// TwinCAT 3 PLC project CNM_AssertionInterfaceTests
// Title: CNM_AssertionInterfaceTests
// Company: ekvip automation GmbH
// Author: boez & ajum
// ProjectVersion: 1.2.0.6
// Description: dirty desperate Foo bar baz run it or go to jail
// ProgramVersion: 3.1.4026.19
// libraries:
//   CNM_AbstractObject, * (ekvip automation GmbH)
//   CNM_AssertionInterfaces, * (ekvip automation GmbH)
//   CNM_ReturnTypes, * (ekvip automation GmbH)
//   CNM_UnicodeUtilities, * (ekvip automation GmbH)
//   Tc2_CncBase, * (Beckhoff Automation GmbH)
//   Tc2_CncHli, * (Beckhoff Automation GmbH)
//   Tc2_Standard, * (Beckhoff Automation GmbH)
//   Tc2_System, * (Beckhoff Automation GmbH)
//   Tc2_Utilities, * (Beckhoff Automation GmbH)
//   Tc3_Module, * (Beckhoff Automation GmbH)
//   TcUnit, * (www.tcunit.org)
// project tree:
//   AssertionTester/AssertionResult/interfaces/ IAssertorContainer.TcIO
//   AssertionTester/AssertionTests/BinaryAssertions/classes/ BinaryAssertionsTests.TcPOU
//   AssertionTester/AssertionTests/BitNumberAssertions/classes/ ByteAssertionTests.TcPOU, XWordAssertionTests.TcPOU, LWordAssertionTests.TcPOU, DWordAssertionTests.TcPOU, WordAssertionTests.TcPOU, XWordAssertionTests.TcPOU
//   AssertionTester/AssertionTests/classes/ AbstractAssertorTest.TcPOU
//   AssertionTester/AssertionTests/DateTimeAssertions/classes/ DTAssertionTests.TcPOU, DateAssertionTests.TcPOU, LDateAssertionTests.TcPOU, LDTAssertionTests.TcPOU, LTODAssertionTests.TcPOU, TODAssertionTests.TcPOU
//   AssertionTester/AssertionTests/FloatAssertions/classes/ LRealAssertionTests.TcPOU, RealAssertionTests.TcPOU
//   AssertionTester/AssertionTests/FloatAssertions/types/structs/ LRealTestParameter.TcDUT (not stored)
//   AssertionTester/AssertionTests/IntegerAssertions/classes/ DintAssertionTests.TcPOU, IntAssertionTests.TcPOU, LintAssertionTests.TcPOU, SintAssertionTests.TcPOU, UdintAssertionTests.TcPOU, UintAssertionTests.TcPOU, UlintAssertionTests.TcPOU, UsintAssertionTests.TcPOU, UxintAssertionTests.TcPOU, XintAssertionTests.TcPOU
//   AssertionTester/AssertionTests/ObjectAssertions/classes/internal/ ConcreteObject.TcPOU, DWordValue.TcPOU, ReverseOrderComparator.TcPOU
//   AssertionTester/AssertionTests/ObjectAssertions/classes/ ObjectAssertionsTests.TcPOU
//   AssertionTester/AssertionTests/ObjectAssertions/interfaces/ IDWord.TcIO
//   AssertionTester/AssertionTests/PointerAssertions/classes/ PointerAssertionsTests.TcPOU
//   AssertionTester/AssertionTests/StringAssertions/classes/ UnicodeUtf16StringAssertionTests.TcPOU, UnicodeUtf8StringAssertionTests.TcPOU, Windows125xStringAssertionTests.TcPOU
//   AssertionTester/AssertionTests/TimeAssertions/classes/ LTimeAssertionsTests.TcPOU, TimeAssertionsTests.TcPOU
//   AssertionTester/classes/ AssertionTester.TcPOU
//   AssertionTester/interfaces/ IAttachAssertorContainer.TcIO
//   Project Information/ F_GetCompany.TcPOU, F_GetTitle.TcPOU, F_GetVersion.TcPOU
//   Version/ Global_Version.TcGVL

// ---- Version/Global_Version.TcGVL
{attribute 'TcGenerated'}
{attribute 'no-analysis'}
{attribute 'linkalways'}
// This function has been automatically generated from the project information.
VAR_GLOBAL CONSTANT
	{attribute 'const_non_replaced'}
	stLibVersion_CNM_AssertionInterfaceTests : ST_LibVersion := (iMajor := 1, iMinor := 2, iBuild := 0, iRevision := 6, nFlags := 0, sVersion := '1.2.0.6');
END_VAR

// ---- AssertionTester/AssertionResult/interfaces/IAssertorContainer.TcIO
(*

short summary
=============
An assertion is handled internally, and there is no common way to determine if an assertion was wrong.
This interface is just a helper to build containers to test assertions in a unified way.

.. <legal notes>

legal notes
=================
| SPDX-FileCopyrightText: © 2023 ekvip automation GmbH <info@ekvip.de>
| SPDX-License-Identifier: Apache-2.0
| For details check: Apache-2.0_

.. _Apache-2.0: https://www.apache.org/licenses/LICENSE-2.0

.. </legal notes>

properties
==========

*)

INTERFACE IAssertorContainer //EXTENDS CNM_AbstractObject.IObject

PROPERTY assertor :CNM_AssertionInterfaces.IAssertor
GET
END_GET
END_PROPERTY

METHOD resetAssertor
VAR_INPUT
END_VAR
END_METHOD

(*

short summary
=============
This property is used by the tests to determine if the assertion was right or wrong (getter)

.. <legal notes>

legal notes
=================
| SPDX-FileCopyrightText: © 2022 ekvip automation GmbH <info@ekvip.de>
| SPDX-License-Identifier: Apache-2.0
| For details check: Apache-2.0_

.. _Apache-2.0: https://www.apache.org/licenses/LICENSE-2.0

.. </legal notes>

*)

PROPERTY wasAssertionWrong :BOOL
GET
END_GET
END_PROPERTY

END_INTERFACE

// ---- AssertionTester/AssertionTests/ObjectAssertions/interfaces/IDWord.TcIO
(*

short summary
=============
Interface for DWordValue Class
only needed for ´´__QUERYINTERFACE()´´ in ´´compareTo()´´
.. <legal notes>

legal notes
=================
| SPDX-FileCopyrightText: © 2023 ekvip automation GmbH <info@ekvip.de>
| SPDX-License-Identifier: Apache-2.0
| For details check: Apache-2.0_

.. _Apache-2.0: https://www.apache.org/licenses/LICENSE-2.0

.. </legal notes>

*)

INTERFACE IDWord EXTENDS CNM_AbstractObject.IObject

(*

short summary
=============
value of the DWordValue Class

.. <legal notes>

legal notes
=================
| SPDX-FileCopyrightText: © 2023 ekvip automation GmbH <info@ekvip.de>
| SPDX-License-Identifier: Apache-2.0
| For details check: Apache-2.0_

.. _Apache-2.0: https://www.apache.org/licenses/LICENSE-2.0

.. </legal notes>

*)

PROPERTY value : DWORD
GET
END_GET
SET
END_SET
END_PROPERTY

END_INTERFACE

// ---- AssertionTester/interfaces/IAttachAssertorContainer.TcIO
(*

short summary
=============

.. <legal notes>

legal notes
=================
| SPDX-FileCopyrightText: © 2023 ekvip automation GmbH <info@ekvip.de>
| SPDX-License-Identifier: Apache-2.0
| For details check: Apache-2.0_

.. _Apache-2.0: https://www.apache.org/licenses/LICENSE-2.0

.. </legal notes>

*)

INTERFACE IAttachAssertorContainer EXTENDS  __SYSTEM.IQueryInterface

(*

short summary
=============

.. <legal notes>

legal notes
=================
| SPDX-FileCopyrightText: © 2023 ekvip automation GmbH <info@ekvip.de>
| SPDX-License-Identifier: Apache-2.0
| For details check: Apache-2.0_

.. _Apache-2.0: https://www.apache.org/licenses/LICENSE-2.0

.. </legal notes>

*)

PROPERTY attachAssertorContainer : IAssertorContainer
SET
END_SET
END_PROPERTY

END_INTERFACE

// ---- AssertionTester/AssertionTests/BinaryAssertions/classes/BinaryAssertionsTests.TcPOU
(*

short summary
==================
This class tests all methods of binary assertions
with various combinations of inputs and checks expected 
outputs are satisfied or not

.. <legal notes>

legal notes
=================
| SPDX-FileCopyrightText: © 2022 ekvip automation GmbH <info@ekvip.de>
| SPDX-License-Identifier: Apache-2.0
| For details check: Apache-2.0_

.. _Apache-2.0: https://www.apache.org/licenses/LICENSE-2.0

.. </legal notes>

methods and properties
======================

*)

FUNCTION_BLOCK BinaryAssertionsTests EXTENDS AbstractAssertorTest
VAR_INPUT
	(* shall be not set, because this is for the null pointer edge case tests *)
	NULL :ANY;
END_VAR
VAR
	(* boolean value TRUE *)
	BOOLEAN_TRUE							:BOOL := TRUE;
	(* boolean value FALSE *)
	BOOLEAN_FALSE							:BOOL := FALSE;
	(* long word value one *)
	LWORD_WITH_VALUE_1						:LWORD := 16#0000_0000_0000_0000_0000_0000_0000_0001;
	(* word value 255 *)
	ALL_BITS_SET_AT_LOW_BYTE				:WORD := 16#00FF;
	(* double word vaule 255 *)
	ALL_BITS_SET_AT_LOW_BYTE_DWORD			:DWORD := 16#0000_00FF;
	(* double word value 16#FF00_FF00 *)
	NO_BITS_SET_AT_MID_BYTES				:DWORD := 16#FF00_00FF;
	(* byte array [0..299] all zero *)
	BYTE_ARRAY_ALL_BYTES_ZERO				:ARRAY[0..299] OF BYTE := [300(0)];
	(* byte array [0..299] 100 zero, 100 16#FF, 100 zero *)
	BYTE_ARRAY_MID_BYTES_FF_ONLY			:ARRAY[0..299] OF BYTE := [100(0),100(16#FF),100(0)];
	(* byte array with two dimensions [0..2][0..99] all zero *)
	ARRAY_OF_BYTE_ARRAY_ALL_BYTES_ZERO		:ARRAY[0..2] OF ARRAY[0..99] OF BYTE := [[100(0)],[100(0)],[100(0)]];	
END_VAR
VAR CONSTANT	
	(* prefix to unify the test names *)
	TEST_NAME_PREFIX						:STRING := 'assert.binary.';
END_VAR

THIS^.runIsEqualToTests();
THIS^.runIsNotEqualToTests();
THIS^.runIsGreaterThanTests();
THIS^.runIsLessThanTests();

(*

short summary
==================
This test method is a helper function to create a unified test name

.. <legal notes>

legal notes
=================
| SPDX-FileCopyrightText: © 2022 ekvip automation GmbH <info@ekvip.de>
| SPDX-License-Identifier: Apache-2.0
| For details check: Apache-2.0_

.. _Apache-2.0: https://www.apache.org/licenses/LICENSE-2.0

.. </legal notes>

parameters
==========

*)

METHOD PROTECTED getTestNameFor :Tc2_System.T_MaxString
VAR_INPUT
	(* name of the method to test, to create a unified test name *)
	nameOfMethodToTest	:Tc2_System.T_MaxString;
END_VAR
getTestNameFor := Tc2_Standard.CONCAT(THIS^.TEST_NAME_PREFIX, nameOfMethodToTest);
END_METHOD

(*

short summary
==================
This test method tests ``assert.binary.isEqualTo``
method of CNM_AssertionInterfaces library with various inputs

.. <legal notes>

legal notes
=================
| SPDX-FileCopyrightText: © 2022 ekvip automation GmbH <info@ekvip.de>
| SPDX-License-Identifier: Apache-2.0
| For details check: Apache-2.0_

.. _Apache-2.0: https://www.apache.org/licenses/LICENSE-2.0

.. </legal notes>

*)

METHOD runIsEqualToTests
RETURN (NOT TcUnit.TEST_ORDERED(THIS^.getTestNameFor('isEqualTo')));

THIS^.testIsEqualTo(
	data			:= THIS^.BOOLEAN_FALSE,
	dataToCompare	:= THIS^.BOOLEAN_FALSE,
	assertionIsWrong:= FALSE,
	testDataInfo	:= 'data is a boolean FALSE, dataToCompare is a aboolean FALSE'
);

THIS^.testIsEqualTo(
	data			:= THIS^.BOOLEAN_TRUE,
	dataToCompare	:= THIS^.BOOLEAN_FALSE,
	assertionIsWrong:= TRUE,
	testDataInfo	:= 'data is a boolean TRUE, dataToCompare is a boolean FALSE'
);

THIS^.testIsEqualTo(
	data			:= THIS^.BOOLEAN_TRUE,
	dataToCompare	:= NULL,
	assertionIsWrong:= TRUE,
	testDataInfo	:= 'data is a boolean TRUE, dataToCompare is null'
);

THIS^.testIsEqualTo(
	data			:= NULL,
	dataToCompare	:= NULL,
	assertionIsWrong:= FALSE,
	testDataInfo	:= 'data is null, dataToCompare is null'
);

THIS^.testIsEqualTo(
	data			:= THIS^.BYTE_ARRAY_ALL_BYTES_ZERO,
	dataToCompare	:= THIS^.BOOLEAN_FALSE,
	assertionIsWrong:= FALSE,
	testDataInfo	:= 'data is a byte array [300(0)], dataToCompare is a boolean FALSE'
);

THIS^.testIsEqualTo(
	data			:= THIS^.BYTE_ARRAY_ALL_BYTES_ZERO,
	dataToCompare	:= THIS^.ARRAY_OF_BYTE_ARRAY_ALL_BYTES_ZERO,
	assertionIsWrong:= FALSE,
	testDataInfo	:= 'data is a byte array [300(0)], dataToCompare is a byte array [[100(0)],[100(0)],[100(0)]]'
);

THIS^.testIsEqualTo(
	data			:= THIS^.BYTE_ARRAY_MID_BYTES_FF_ONLY,
	dataToCompare	:= THIS^.ARRAY_OF_BYTE_ARRAY_ALL_BYTES_ZERO,
	assertionIsWrong:= TRUE,
	testDataInfo	:= 'data is a byte array [100(0),100(16#FF),100(0)], dataToCompare is a byte array [[100(0)],[100(0)],[100(0)]]'
);

THIS^.testIsEqualTo(
	data			:= THIS^.ALL_BITS_SET_AT_LOW_BYTE,
	dataToCompare	:= THIS^.ALL_BITS_SET_AT_LOW_BYTE_DWORD,
	assertionIsWrong:= FALSE,
	testDataInfo	:= 'data is a word 16#00FF, dataToCompare is dword 16#0000_00FF'
);

THIS^.testIsEqualTo(
	data			:= THIS^.ALL_BITS_SET_AT_LOW_BYTE_DWORD,
	dataToCompare	:= THIS^.ALL_BITS_SET_AT_LOW_BYTE,
	assertionIsWrong:= FALSE,
	testDataInfo	:= 'data is a dword 16#0000_00FF, dataToCompare is word 16#00FF'
);

THIS^.testIsEqualTo(
	data			:= THIS^.ALL_BITS_SET_AT_LOW_BYTE,
	dataToCompare	:= THIS^.NO_BITS_SET_AT_MID_BYTES,
	assertionIsWrong:= TRUE,
	testDataInfo	:= 'data is a word 16#00FF, dataToCompare is dword 16#FF00_00FF'
);

THIS^.testIsEqualTo(
	data			:= THIS^.NO_BITS_SET_AT_MID_BYTES,
	dataToCompare	:= THIS^.ALL_BITS_SET_AT_LOW_BYTE,
	assertionIsWrong:= TRUE,
	testDataInfo	:= 'data is a dword 16#FF00_00FF, dataToCompare is word 16#00FF'
);

THIS^.testIsEqualTo(
	data			:= THIS^.LWORD_WITH_VALUE_1,
	dataToCompare	:= THIS^.BOOLEAN_TRUE,
	assertionIsWrong:= FALSE,
	testDataInfo	:= 'data is a lword 16#0000_0000_0000_0000_0000_0000_0000_0001, dataToCompare is bool TRUE'
);

THIS^.testIsEqualTo(
	data			:= THIS^.LWORD_WITH_VALUE_1,
	dataToCompare	:= THIS^.BOOLEAN_FALSE,
	assertionIsWrong:= TRUE,
	testDataInfo	:= 'data is a lword 16#0000_0000_0000_0000_0000_0000_0000_0001, dataToCompare is bool FALSE'
);

TcUnit.TEST_FINISHED();
END_METHOD

(*

short summary
==================
This test method tests ``assert.binary.isGreaterThan``
method of CNM_AssertionInterfaces library with various inputs

.. <legal notes>

legal notes
=================
| SPDX-FileCopyrightText: © 2022 ekvip automation GmbH <info@ekvip.de>
| SPDX-License-Identifier: Apache-2.0
| For details check: Apache-2.0_

.. _Apache-2.0: https://www.apache.org/licenses/LICENSE-2.0

.. </legal notes>

*)

METHOD runIsGreaterThanTests
RETURN (NOT TcUnit.TEST_ORDERED(THIS^.getTestNameFor('isGreaterThan')));

THIS^.testIsGreaterThan(
	data			:= THIS^.BOOLEAN_FALSE,
	dataToCompare	:= THIS^.BOOLEAN_FALSE,
	assertionIsWrong:= TRUE,
	testDataInfo	:= 'data is a boolean FALSE, dataToCompare is a aboolean FALSE'
);

THIS^.testIsGreaterThan(
	data			:= THIS^.BOOLEAN_TRUE,
	dataToCompare	:= THIS^.BOOLEAN_FALSE,
	assertionIsWrong:= FALSE,
	testDataInfo	:= 'data is a boolean TRUE, dataToCompare is a boolean FALSE'
);

THIS^.testIsGreaterThan(
	data			:= THIS^.BOOLEAN_TRUE,
	dataToCompare	:= NULL,
	assertionIsWrong:= FALSE,
	testDataInfo	:= 'data is a boolean TRUE, dataToCompare is null'
);

THIS^.testIsGreaterThan(
	data			:= NULL,
	dataToCompare	:= NULL,
	assertionIsWrong:= TRUE,
	testDataInfo	:= 'data is null, dataToCompare is null'
);

THIS^.testIsGreaterThan(
	data			:= THIS^.BYTE_ARRAY_ALL_BYTES_ZERO,
	dataToCompare	:= THIS^.BOOLEAN_FALSE,
	assertionIsWrong:= TRUE,
	testDataInfo	:= 'data is a byte array [300(0)], dataToCompare is a boolean FALSE'
);

THIS^.testIsGreaterThan(
	data			:= THIS^.BYTE_ARRAY_ALL_BYTES_ZERO,
	dataToCompare	:= THIS^.ARRAY_OF_BYTE_ARRAY_ALL_BYTES_ZERO,
	assertionIsWrong:= TRUE,
	testDataInfo	:= 'data is a byte array [300(0)], dataToCompare is a byte array [[100(0)],[100(0)],[100(0)]]'
);

THIS^.testIsGreaterThan(
	data			:= THIS^.BYTE_ARRAY_MID_BYTES_FF_ONLY,
	dataToCompare	:= THIS^.ARRAY_OF_BYTE_ARRAY_ALL_BYTES_ZERO,
	assertionIsWrong:= FALSE,
	testDataInfo	:= 'data is a byte array [100(0),100(16#FF),100(0)], dataToCompare is a byte array [[100(0)],[100(0)],[100(0)]]'
);

THIS^.testIsGreaterThan(
	data			:= THIS^.ALL_BITS_SET_AT_LOW_BYTE,
	dataToCompare	:= THIS^.ALL_BITS_SET_AT_LOW_BYTE_DWORD,
	assertionIsWrong:= TRUE,
	testDataInfo	:= 'data is a word 16#00FF, dataToCompare is dword 16#0000_00FF'
);

THIS^.testIsGreaterThan(
	data			:= THIS^.ALL_BITS_SET_AT_LOW_BYTE_DWORD,
	dataToCompare	:= THIS^.ALL_BITS_SET_AT_LOW_BYTE,
	assertionIsWrong:= TRUE,
	testDataInfo	:= 'data is a dword 16#0000_00FF, dataToCompare is word 16#00FF'
);

THIS^.testIsGreaterThan(
	data			:= THIS^.ALL_BITS_SET_AT_LOW_BYTE,
	dataToCompare	:= THIS^.NO_BITS_SET_AT_MID_BYTES,
	assertionIsWrong:= TRUE,
	testDataInfo	:= 'data is a word 16#00FF, dataToCompare is dword 16#FF00_00FF'
);

THIS^.testIsGreaterThan(
	data			:= THIS^.NO_BITS_SET_AT_MID_BYTES,
	dataToCompare	:= THIS^.ALL_BITS_SET_AT_LOW_BYTE,
	assertionIsWrong:= FALSE,
	testDataInfo	:= 'data is a dword 16#FF00_00FF, dataToCompare is word 16#00FF'
);

THIS^.testIsGreaterThan(
	data			:= THIS^.LWORD_WITH_VALUE_1,
	dataToCompare	:= THIS^.BOOLEAN_TRUE,
	assertionIsWrong:= TRUE,
	testDataInfo	:= 'data is a lword 16#0000_0000_0000_0000_0000_0000_0000_0001, dataToCompare is bool TRUE'
);

THIS^.testIsGreaterThan(
	data			:= THIS^.LWORD_WITH_VALUE_1,
	dataToCompare	:= THIS^.BOOLEAN_FALSE,
	assertionIsWrong:= FALSE,
	testDataInfo	:= 'data is a lword 16#0000_0000_0000_0000_0000_0000_0000_0001, dataToCompare is bool FALSE'
);

THIS^.testIsGreaterThan(
	data			:= THIS^.BOOLEAN_TRUE,
	dataToCompare	:= THIS^.LWORD_WITH_VALUE_1,
	assertionIsWrong:= TRUE,
	testDataInfo	:= 'data is a bool TRUE, dataToCompare is bool 16#0000_0000_0000_0000_0000_0000_0000_0001'
);

THIS^.testIsGreaterThan(
	data			:= THIS^.BOOLEAN_FALSE,
	dataToCompare	:= THIS^.LWORD_WITH_VALUE_1,
	assertionIsWrong:= TRUE,
	testDataInfo	:= 'data is a bool FALSE, dataToCompare is bool 16#0000_0000_0000_0000_0000_0000_0000_0001'
);

TcUnit.TEST_FINISHED();
END_METHOD

(*

short summary
==================
This test method tests ``assert.binary.isLessThan``
method of CNM_AssertionInterfaces library with various inputs

.. <legal notes>

legal notes
=================
| SPDX-FileCopyrightText: © 2022 ekvip automation GmbH <info@ekvip.de>
| SPDX-License-Identifier: Apache-2.0
| For details check: Apache-2.0_

.. _Apache-2.0: https://www.apache.org/licenses/LICENSE-2.0

.. </legal notes>

*)

METHOD runIsLessThanTests
RETURN (NOT TcUnit.TEST_ORDERED(THIS^.getTestNameFor('isLessThan')));

THIS^.testIsLessThan(
	data			:= THIS^.BOOLEAN_FALSE,
	dataToCompare	:= THIS^.BOOLEAN_FALSE,
	assertionIsWrong:= TRUE,
	testDataInfo	:= 'data is a boolean FALSE, dataToCompare is a aboolean FALSE'
);

THIS^.testIsLessThan(
	data			:= THIS^.BOOLEAN_TRUE,
	dataToCompare	:= THIS^.BOOLEAN_FALSE,
	assertionIsWrong:= TRUE,
	testDataInfo	:= 'data is a boolean TRUE, dataToCompare is a boolean FALSE'
);

THIS^.testIsLessThan(
	data			:= THIS^.BOOLEAN_FALSE,
	dataToCompare	:= THIS^.BOOLEAN_TRUE,
	assertionIsWrong:= FALSE,
	testDataInfo	:= 'data is a boolean FALSE, dataToCompare is a boolean TRUE'
);

THIS^.testIsLessThan(
	data			:= THIS^.BOOLEAN_TRUE,
	dataToCompare	:= NULL,
	assertionIsWrong:= TRUE,
	testDataInfo	:= 'data is a boolean TRUE, dataToCompare is null'
);

THIS^.testIsLessThan(
	data			:= NULL,
	dataToCompare	:= THIS^.BOOLEAN_TRUE,
	assertionIsWrong:= FALSE,
	testDataInfo	:= 'data is null, dataToCompare is a boolean TRUE'
);

THIS^.testIsLessThan(
	data			:= NULL,
	dataToCompare	:= NULL,
	assertionIsWrong:= TRUE,
	testDataInfo	:= 'data is null, dataToCompare is null'
);

THIS^.testIsLessThan(
	data			:= THIS^.BYTE_ARRAY_ALL_BYTES_ZERO,
	dataToCompare	:= THIS^.BOOLEAN_FALSE,
	assertionIsWrong:= TRUE,
	testDataInfo	:= 'data is a byte array [300(0)], dataToCompare is a boolean FALSE'
);

THIS^.testIsLessThan(
	data			:= THIS^.BYTE_ARRAY_ALL_BYTES_ZERO,
	dataToCompare	:= THIS^.ARRAY_OF_BYTE_ARRAY_ALL_BYTES_ZERO,
	assertionIsWrong:= TRUE,
	testDataInfo	:= 'data is a byte array [300(0)], dataToCompare is a byte array [[100(0)],[100(0)],[100(0)]]'
);

THIS^.testIsLessThan(
	data			:= THIS^.ARRAY_OF_BYTE_ARRAY_ALL_BYTES_ZERO,
	dataToCompare	:= THIS^.BYTE_ARRAY_ALL_BYTES_ZERO,
	assertionIsWrong:= TRUE,
	testDataInfo	:= 'data is a byte array [100(0),100(0),100(0)], dataToCompare is a byte array [300(0)]'
);

THIS^.testIsLessThan(
	data			:= THIS^.BYTE_ARRAY_MID_BYTES_FF_ONLY,
	dataToCompare	:= THIS^.ARRAY_OF_BYTE_ARRAY_ALL_BYTES_ZERO,
	assertionIsWrong:= TRUE,
	testDataInfo	:= 'data is a byte array [100(0),100(16#FF),100(0)], dataToCompare is a byte array [[100(0)],[100(0)],[100(0)]]'
);

THIS^.testIsLessThan(
	data			:= THIS^.ARRAY_OF_BYTE_ARRAY_ALL_BYTES_ZERO,
	dataToCompare	:= THIS^.BYTE_ARRAY_MID_BYTES_FF_ONLY,
	assertionIsWrong:= FALSE,
	testDataInfo	:= 'data is a byte array [[100(0)],[100(0)],[100(0)]], dataToCompare is a byte array [100(0),100(16#FF),100(0)]'
);

THIS^.testIsLessThan(
	data			:= THIS^.ALL_BITS_SET_AT_LOW_BYTE_DWORD,
	dataToCompare	:= THIS^.ALL_BITS_SET_AT_LOW_BYTE,
	assertionIsWrong:= TRUE,
	testDataInfo	:= 'data is a dword 16#0000_00FF, dataToCompare is word 16#00FF'
);

THIS^.testIsLessThan(
	data			:= THIS^.ALL_BITS_SET_AT_LOW_BYTE,
	dataToCompare	:= THIS^.NO_BITS_SET_AT_MID_BYTES,
	assertionIsWrong:= FALSE,
	testDataInfo	:= 'data is a word 16#00FF, dataToCompare is dword 16#FF00_00FF'
);

THIS^.testIsLessThan(
	data			:= THIS^.NO_BITS_SET_AT_MID_BYTES,
	dataToCompare	:= THIS^.ALL_BITS_SET_AT_LOW_BYTE,
	assertionIsWrong:= TRUE,
	testDataInfo	:= 'data is a dword 16#FF00_00FF, dataToCompare is word 16#00FF'
);

THIS^.testIsLessThan(
	data			:= THIS^.LWORD_WITH_VALUE_1,
	dataToCompare	:= THIS^.BOOLEAN_TRUE,
	assertionIsWrong:= TRUE,
	testDataInfo	:= 'data is a lword 16#0000_0000_0000_0000_0000_0000_0000_0001, dataToCompare is bool TRUE'
);

THIS^.testIsLessThan(
	data			:= THIS^.LWORD_WITH_VALUE_1,
	dataToCompare	:= THIS^.BOOLEAN_FALSE,
	assertionIsWrong:= TRUE,
	testDataInfo	:= 'data is a lword 16#0000_0000_0000_0000_0000_0000_0000_0001, dataToCompare is bool FALSE'
);

THIS^.testIsLessThan(
	data			:= THIS^.BOOLEAN_TRUE,
	dataToCompare	:= THIS^.LWORD_WITH_VALUE_1,
	assertionIsWrong:= TRUE,
	testDataInfo	:= 'data is a bool TRUE, dataToCompare is bool 16#0000_0000_0000_0000_0000_0000_0000_0001'
);

THIS^.testIsLessThan(
	data			:= THIS^.BOOLEAN_FALSE,
	dataToCompare	:= THIS^.LWORD_WITH_VALUE_1,
	assertionIsWrong:= FALSE,
	testDataInfo	:= 'data is a bool FALSE, dataToCompare is bool 16#0000_0000_0000_0000_0000_0000_0000_0001'
);

TcUnit.TEST_FINISHED();
END_METHOD

(*

short summary
==================
This test method tests ``assert.binary.isNotEqualTo``
method of CNM_AssertionInterfaces library with various inputs

.. <legal notes>

legal notes
=================
| SPDX-FileCopyrightText: © 2022 ekvip automation GmbH <info@ekvip.de>
| SPDX-License-Identifier: Apache-2.0
| For details check: Apache-2.0_

.. _Apache-2.0: https://www.apache.org/licenses/LICENSE-2.0

.. </legal notes>

*)

METHOD runIsNotEqualToTests
RETURN (NOT TcUnit.TEST_ORDERED(THIS^.getTestNameFor('isNotEqualTo')));

THIS^.testIsNotEqualTo(
	data			:= THIS^.BOOLEAN_FALSE,
	dataToCompare	:= THIS^.BOOLEAN_FALSE,
	assertionIsWrong:= TRUE,
	testDataInfo	:= 'data is a boolean FALSE, dataToCompare is a aboolean FALSE'
);

THIS^.testIsNotEqualTo(
	data			:= THIS^.BOOLEAN_TRUE,
	dataToCompare	:= THIS^.BOOLEAN_FALSE,
	assertionIsWrong:= FALSE,
	testDataInfo	:= 'data is a boolean TRUE, dataToCompare is a boolean FALSE'
);

THIS^.testIsNotEqualTo(
	data			:= THIS^.BOOLEAN_TRUE,
	dataToCompare	:= NULL,
	assertionIsWrong:= FALSE,
	testDataInfo	:= 'data is a boolean TRUE, dataToCompare is null'
);

THIS^.testIsNotEqualTo(
	data			:= NULL,
	dataToCompare	:= NULL,
	assertionIsWrong:= TRUE,
	testDataInfo	:= 'data is null, dataToCompare is null'
);

THIS^.testIsNotEqualTo(
	data			:= THIS^.BYTE_ARRAY_ALL_BYTES_ZERO,
	dataToCompare	:= THIS^.BOOLEAN_FALSE,
	assertionIsWrong:= TRUE,
	testDataInfo	:= 'data is a byte array [300(0)], dataToCompare is a boolean FALSE'
);

THIS^.testIsNotEqualTo(
	data			:= THIS^.BYTE_ARRAY_ALL_BYTES_ZERO,
	dataToCompare	:= THIS^.ARRAY_OF_BYTE_ARRAY_ALL_BYTES_ZERO,
	assertionIsWrong:= TRUE,
	testDataInfo	:= 'data is a byte array [300(0)], dataToCompare is a byte array [[100(0)],[100(0)],[100(0)]]'
);

THIS^.testIsNotEqualTo(
	data			:= THIS^.BYTE_ARRAY_MID_BYTES_FF_ONLY,
	dataToCompare	:= THIS^.ARRAY_OF_BYTE_ARRAY_ALL_BYTES_ZERO,
	assertionIsWrong:= FALSE,
	testDataInfo	:= 'data is a byte array [100(0),100(16#FF),100(0)], dataToCompare is a byte array [[100(0)],[100(0)],[100(0)]]'
);

THIS^.testIsNotEqualTo(
	data			:= THIS^.ALL_BITS_SET_AT_LOW_BYTE,
	dataToCompare	:= THIS^.ALL_BITS_SET_AT_LOW_BYTE_DWORD,
	assertionIsWrong:= TRUE,
	testDataInfo	:= 'data is a word 16#00FF, dataToCompare is dword 16#0000_00FF'
);

THIS^.testIsNotEqualTo(
	data			:= THIS^.ALL_BITS_SET_AT_LOW_BYTE_DWORD,
	dataToCompare	:= THIS^.ALL_BITS_SET_AT_LOW_BYTE,
	assertionIsWrong:= TRUE,
	testDataInfo	:= 'data is a dword 16#0000_00FF, dataToCompare is word 16#00FF'
);

THIS^.testIsNotEqualTo(
	data			:= THIS^.ALL_BITS_SET_AT_LOW_BYTE,
	dataToCompare	:= THIS^.NO_BITS_SET_AT_MID_BYTES,
	assertionIsWrong:= FALSE,
	testDataInfo	:= 'data is a word 16#00FF, dataToCompare is dword 16#FF00_00FF'
);

THIS^.testIsNotEqualTo(
	data			:= THIS^.NO_BITS_SET_AT_MID_BYTES,
	dataToCompare	:= THIS^.ALL_BITS_SET_AT_LOW_BYTE,
	assertionIsWrong:= FALSE,
	testDataInfo	:= 'data is a dword 16#FF00_00FF, dataToCompare is word 16#00FF'
);

THIS^.testIsNotEqualTo(
	data			:= THIS^.LWORD_WITH_VALUE_1,
	dataToCompare	:= THIS^.BOOLEAN_TRUE,
	assertionIsWrong:= TRUE,
	testDataInfo	:= 'data is a lword 16#0000_0000_0000_0000_0000_0000_0000_0001, dataToCompare is bool TRUE'
);

THIS^.testIsNotEqualTo(
	data			:= THIS^.LWORD_WITH_VALUE_1,
	dataToCompare	:= THIS^.BOOLEAN_FALSE,
	assertionIsWrong:= FALSE,
	testDataInfo	:= 'data is a lword 16#0000_0000_0000_0000_0000_0000_0000_0001, dataToCompare is bool FALSE'
);

TcUnit.TEST_FINISHED();
END_METHOD

(*

short summary
==================
This test method tests ``assert.binary.isEqualTo``
method of CNM_AssertionInterfaces library, 
it provides the possibility to handover test data via parameter 


.. <legal notes>

legal notes
=================
| SPDX-FileCopyrightText: © 2022 ekvip automation GmbH <info@ekvip.de>
| SPDX-License-Identifier: Apache-2.0
| For details check: Apache-2.0_

.. _Apache-2.0: https://www.apache.org/licenses/LICENSE-2.0

.. </legal notes>

parameters
==========

*)

METHOD testIsEqualTo 
VAR_INPUT
	(* for the test it's the parameter ``data`` *)
	data				:ANY;
	(* for the test it's the parameter ``dataToCompare`` *)
	dataToCompare		:ANY;
	(* just the expectation if the assertion to test must be worng or true *)
	assertionIsWrong	:BOOL;
	(* info string what the test does *)
	testDataInfo		:Tc2_System.T_MaxString;
END_VAR
VAR
	(* contains the format string for the test message *)
	message	:Tc2_System.T_MaxString;
END_VAR
THIS^.assertorContainer.resetAssertor();

message := SEL(
	assertionIsWrong,
	Tc2_Standard.CONCAT(testDataInfo, ' assertion must be TRUE'),
	Tc2_Standard.CONCAT(testDataInfo, ' assertion must be FALSE')
);

THIS^.assertorContainer.assertor.assert.binary.isEqualTo(
	data := data,
	dataToCompare := dataToCompare,
	message := ''
);

THIS^.AssertEquals_BOOL(
	Expected 	:= assertionIsWrong,
	Actual 		:= THIS^.assertorContainer.wasAssertionWrong,
	Message 	:= message
);
END_METHOD

(*

short summary
==================
This test method tests ``assert.binary.isGreaterThan``
method of CNM_AssertionInterfaces library, 
it provides the possibility to handover test data via parameter 


.. <legal notes>

legal notes
=================
| SPDX-FileCopyrightText: © 2022 ekvip automation GmbH <info@ekvip.de>
| SPDX-License-Identifier: Apache-2.0
| For details check: Apache-2.0_

.. _Apache-2.0: https://www.apache.org/licenses/LICENSE-2.0

.. </legal notes>

parameters
==========

*)

METHOD testIsGreaterThan 
VAR_INPUT
	(* for the test it's the parameter ``data`` *)
	data				:ANY;
	(* for the test it's the parameter ``dataToCompare`` *)
	dataToCompare		:ANY;
	(* just the expectation if the assertion to test must be worng or true *)
	assertionIsWrong	:BOOL;
	(* info string what the test does *)
	testDataInfo		:Tc2_System.T_MaxString;
END_VAR
VAR
	(* contains the format string for the test message *)
	message	:Tc2_System.T_MaxString;
END_VAR
THIS^.assertorContainer.resetAssertor();

message := SEL(
	assertionIsWrong,
	Tc2_Standard.CONCAT(testDataInfo, ' assertion must be TRUE'),
	Tc2_Standard.CONCAT(testDataInfo, ' assertion must be FALSE')
);

THIS^.assertorContainer.assertor.assert.binary.isGreaterThan(
	data := data,
	dataToCompare := dataToCompare,
	message := ''
);

THIS^.AssertEquals_BOOL(
	Expected 	:= assertionIsWrong,
	Actual 		:= THIS^.assertorContainer.wasAssertionWrong,
	Message 	:= message
);
END_METHOD

(*

short summary
==================
This test method tests ``assert.binary.isLessThan``
method of CNM_AssertionInterfaces library, 
it provides the possibility to handover test data via parameter 


.. <legal notes>

legal notes
=================
| SPDX-FileCopyrightText: © 2022 ekvip automation GmbH <info@ekvip.de>
| SPDX-License-Identifier: Apache-2.0
| For details check: Apache-2.0_

.. _Apache-2.0: https://www.apache.org/licenses/LICENSE-2.0

.. </legal notes>

parameters
==========

*)

METHOD testIsLessThan 
VAR_INPUT
	(* for the test it's the parameter ``data`` *)
	data				:ANY;
	(* for the test it's the parameter ``dataToCompare`` *)
	dataToCompare		:ANY;
	(* just the expectation if the assertion to test must be worng or true *)
	assertionIsWrong	:BOOL;
	(* info string what the test does *)
	testDataInfo		:Tc2_System.T_MaxString;
END_VAR
VAR
	(* contains the format string for the test message *)
	message	:Tc2_System.T_MaxString;
END_VAR
THIS^.assertorContainer.resetAssertor();

message := SEL(
	assertionIsWrong,
	Tc2_Standard.CONCAT(testDataInfo, ' assertion must be TRUE'),
	Tc2_Standard.CONCAT(testDataInfo, ' assertion must be FALSE')
);

THIS^.assertorContainer.assertor.assert.binary.isLessThan(
	data := data,
	dataToCompare := dataToCompare,
	message := ''
);

THIS^.AssertEquals_BOOL(
	Expected 	:= assertionIsWrong,
	Actual 		:= THIS^.assertorContainer.wasAssertionWrong,
	Message 	:= message
);
END_METHOD

(*

short summary
==================
This test method tests ``assert.binary.isNotEqualTo``
method of CNM_AssertionInterfaces library, 
it provides the possibility to handover test data via parameter 


.. <legal notes>

legal notes
=================
| SPDX-FileCopyrightText: © 2022 ekvip automation GmbH <info@ekvip.de>
| SPDX-License-Identifier: Apache-2.0
| For details check: Apache-2.0_

.. _Apache-2.0: https://www.apache.org/licenses/LICENSE-2.0

.. </legal notes>

parameters
==========

*)

METHOD testIsNotEqualTo 
VAR_INPUT
	(* for the test it's the parameter ``data`` *)
	data				:ANY;
	(* for the test it's the parameter ``dataToCompare`` *)
	dataToCompare		:ANY;
	(* just the expectation if the assertion to test must be worng or true *)
	assertionIsWrong	:BOOL;
	(* info string what the test does *)
	testDataInfo		:Tc2_System.T_MaxString;
END_VAR
VAR
	(* contains the format string for the test message *)
	message	:Tc2_System.T_MaxString;
END_VAR
THIS^.assertorContainer.resetAssertor();

message := SEL(
	assertionIsWrong,
	Tc2_Standard.CONCAT(testDataInfo, ' assertion must be TRUE'),
	Tc2_Standard.CONCAT(testDataInfo, ' assertion must be FALSE')
);

THIS^.assertorContainer.assertor.assert.binary.isNotEqualTo(
	data := data,
	dataToCompare := dataToCompare,
	message := ''
);

THIS^.AssertEquals_BOOL(
	Expected 	:= assertionIsWrong,
	Actual 		:= THIS^.assertorContainer.wasAssertionWrong,
	Message 	:= message
);
END_METHOD

END_FUNCTION_BLOCK

// ---- AssertionTester/AssertionTests/classes/AbstractAssertorTest.TcPOU
(*

short summary
=============
This provides the possibility for tests to attach an :ref:`ICanAssertWithResult` during the runtime.
All assertion tests are based on it. The late attachment of this class is used by :ref:`AssertionTester.FB_init`.

.. <legal notes>

legal notes
=================
| SPDX-FileCopyrightText: © 2023 ekvip automation GmbH <info@ekvip.de>
| SPDX-License-Identifier: Apache-2.0
| For details check: Apache-2.0_

.. _Apache-2.0: https://www.apache.org/licenses/LICENSE-2.0

.. </legal notes>

properties and methods
=======================

*)

FUNCTION_BLOCK INTERNAL ABSTRACT AbstractAssertorTest EXTENDS TcUnit.FB_TestSuite IMPLEMENTS IAttachAssertorContainer
VAR
	(* container with the concrete assertor which need to be tested *)
	assertorContainer :IAssertorContainer;
END_VAR

(*

summary
==================
helper function to get ``Tc2_Utilities.T_Arg`` for the message formatting


.. <legal notes>

legal notes
=================
| SPDX-FileCopyrightText: © 2022 ekvip automation GmbH <info@ekvip.de>
| SPDX-License-Identifier: Apache-2.0
| For details check: Apache-2.0_

.. _Apache-2.0: https://www.apache.org/licenses/LICENSE-2.0

.. </legal notes>

parameters
==========

*)

METHOD PROTECTED AnyToArg :Tc2_Utilities.T_Arg
VAR_INPUT
	(* just the data which shoud be casted to ``Tc2_Utilities.T_Arg`` *)
	in	:ANY;
END_VAR
VAR
	(* just to store the ``ANY`` without changes *)
	data	:__SYSTEM.AnyType;	
END_VAR
data.diSize := in.diSize;
data.pValue := in.pValue;
data.TypeClass := in.TypeClass;
THIS^.dereferenceAnys(in := data, out => data);
AnyToArg := THIS^.AnyTypeToArg(data);
END_METHOD

(*

summary
==================
helper function to get ``Tc2_Utilities.T_Arg`` for the message formatting


.. <legal notes>

legal notes
=================
| SPDX-FileCopyrightText: © 2022 ekvip automation GmbH <info@ekvip.de>
| SPDX-License-Identifier: Apache-2.0
| For details check: Apache-2.0_

.. _Apache-2.0: https://www.apache.org/licenses/LICENSE-2.0

.. </legal notes>

parameters
==========

*)


METHOD PROTECTED AnyTypeToArg :Tc2_Utilities.T_Arg
VAR_INPUT
	in :__SYSTEM.AnyType;
END_VAR
AnyTypeToArg.cbLen := TO_UDINT(in.diSize);
AnyTypeToArg.pData := in.pValue;
AnyTypeToArg.eType := THIS^.typeClassToArgType(in.TypeClass, AnyTypeToArg.cbLen);
END_METHOD

(*

short summary
=============

.. <legal notes>

legal notes
=================
| SPDX-FileCopyrightText: © 2023 ekvip automation GmbH <info@ekvip.de>
| SPDX-License-Identifier: Apache-2.0
| For details check: Apache-2.0_

.. _Apache-2.0: https://www.apache.org/licenses/LICENSE-2.0

.. </legal notes>

*)


PROPERTY attachAssertorContainer : IAssertorContainer
SET
(*

short summary
=============

.. <legal notes>

legal notes
=================
| SPDX-FileCopyrightText: © 2023 ekvip automation GmbH <info@ekvip.de>
| SPDX-License-Identifier: Apache-2.0
| For details check: Apache-2.0_

.. _Apache-2.0: https://www.apache.org/licenses/LICENSE-2.0

.. </legal notes>

*)

VAR
END_VAR
THIS^.assertorContainer := attachAssertorContainer;
END_SET
END_PROPERTY


METHOD PROTECTED dereferenceAnys
VAR_INPUT
	in :__SYSTEM.AnyType;
END_VAR
VAR_OUTPUT
	out :__SYSTEM.AnyType;	
END_VAR
VAR
	p :POINTER TO __SYSTEM.AnyType;
END_VAR
CASE in.TypeClass OF
__SYSTEM.TYPE_CLASS.TYPE_ANY,  
__SYSTEM.TYPE_CLASS.TYPE_ANYBIT, 
__SYSTEM.TYPE_CLASS.TYPE_ANYDATE,
__SYSTEM.TYPE_CLASS.TYPE_ANYINT,
__SYSTEM.TYPE_CLASS.TYPE_ANYNUM,
__SYSTEM.TYPE_CLASS.TYPE_ANYREAL:
	p := in.pValue;
	p := p^.pValue;
	THIS^.dereferenceAnys(p^, out => out);
ELSE
	out := in;
END_CASE
END_METHOD

(*

short summary
=============

.. <legal notes>

legal notes
=================
| SPDX-FileCopyrightText: © 2023 ekvip automation GmbH <info@ekvip.de>
| SPDX-License-Identifier: Apache-2.0
| For details check: Apache-2.0_

.. _Apache-2.0: https://www.apache.org/licenses/LICENSE-2.0

.. </legal notes>

parameters
==========

*)

METHOD FB_init :BOOL
VAR_INPUT
    bInitRetains	:BOOL; // if TRUE, the retain variables are initialized (warm start / cold start)
    bInCopyCode		:BOOL;  // if TRUE, the instance afterwards gets moved into the copy code (online change)
	classToBeTested :IAssertorContainer;
END_VAR
THIS^.assertorContainer := classToBeTested;
END_METHOD


METHOD PROTECTED typeClassToArgType : Tc2_Utilities.E_ArgType
VAR_INPUT
	typeClass 	:__SYSTEM.TYPE_CLASS;
	size	:UDINT;
END_VAR
VAR CONSTANT
	LENGTH_1_BYTE	:UINT := 1;
	LENGTH_2_BYTE	:UINT := 2;
	LENGTH_4_BYTE	:UINT := 4;
	LENGTH_8_BYTE	:UINT := 8;
END_VAR
CASE typeClass OF
__SYSTEM.TYPE_CLASS.TYPE_BOOL, __SYSTEM.TYPE_CLASS.TYPE_BYTE,
__SYSTEM.TYPE_CLASS.TYPE_BIT:
	typeClassToArgType := Tc2_Utilities.E_ArgType.ARGTYPE_BYTE;
__SYSTEM.TYPE_CLASS.TYPE_WORD:
	typeClassToArgType := Tc2_Utilities.E_ArgType.ARGTYPE_WORD;
__SYSTEM.TYPE_CLASS.TYPE_DWORD:
	typeClassToArgType := Tc2_Utilities.E_ArgType.ARGTYPE_DWORD;
__SYSTEM.TYPE_CLASS.TYPE_LWORD:
	typeClassToArgType := Tc2_Utilities.E_ArgType.ARGTYPE_LWORD;
__SYSTEM.TYPE_CLASS.TYPE_USINT:
	typeClassToArgType := Tc2_Utilities.E_ArgType.ARGTYPE_USINT;
__SYSTEM.TYPE_CLASS.TYPE_SINT:
	typeClassToArgType := Tc2_Utilities.E_ArgType.ARGTYPE_SINT;
__SYSTEM.TYPE_CLASS.TYPE_UINT:
	typeClassToArgType := Tc2_Utilities.E_ArgType.ARGTYPE_UINT;
__SYSTEM.TYPE_CLASS.TYPE_INT:
	typeClassToArgType := Tc2_Utilities.E_ArgType.ARGTYPE_INT;
__SYSTEM.TYPE_CLASS.TYPE_UDINT, __SYSTEM.TYPE_CLASS.TYPE_TIME,
__SYSTEM.TYPE_CLASS.TYPE_DATE, __SYSTEM.TYPE_CLASS.TYPE_DATEANDTIME,
__SYSTEM.TYPE_CLASS.TYPE_TIMEOFDAY:
	typeClassToArgType := Tc2_Utilities.E_ArgType.ARGTYPE_UDINT;
__SYSTEM.TYPE_CLASS.TYPE_DINT:
	typeClassToArgType := Tc2_Utilities.E_ArgType.ARGTYPE_DINT;
__SYSTEM.TYPE_CLASS.TYPE_ULINT, __SYSTEM.TYPE_CLASS.TYPE_LTIME:
		typeClassToArgType := Tc2_Utilities.E_ArgType.ARGTYPE_ULARGE;
__SYSTEM.TYPE_CLASS.TYPE_LINT:
	typeClassToArgType := Tc2_Utilities.E_ArgType.ARGTYPE_LARGE;
__SYSTEM.TYPE_CLASS.TYPE_REAL:
	typeClassToArgType := Tc2_Utilities.E_ArgType.ARGTYPE_REAL;
__SYSTEM.TYPE_CLASS.TYPE_LREAL:
	typeClassToArgType := Tc2_Utilities.E_ArgType.ARGTYPE_LREAL;
__SYSTEM.TYPE_CLASS.TYPE_STRING:
	typeClassToArgType := SEL(
		(size <= SIZEOF(T_MaxString)),
		Tc2_Utilities.E_ArgType.ARGTYPE_UNKNOWN,
		Tc2_Utilities.E_ArgType.ARGTYPE_STRING
	);
__SYSTEM.TYPE_CLASS.TYPE_POINTER, __SYSTEM.TYPE_CLASS.TYPE_REFERENCE:
	typeClassToArgType := SEL(
		(SIZEOF(__XWORD) = SIZEOF(LWORD)),
		Tc2_Utilities.E_ArgType.ARGTYPE_DWORD,
		Tc2_Utilities.E_ArgType.ARGTYPE_LWORD
	);	
__SYSTEM.TYPE_CLASS.TYPE_SUBRANGE, __SYSTEM.TYPE_CLASS.TYPE_ENUM:
	CASE size OF
	LENGTH_1_BYTE: typeClassToArgType := Tc2_Utilities.E_ArgType.ARGTYPE_USINT;
	LENGTH_2_BYTE: typeClassToArgType := Tc2_Utilities.E_ArgType.ARGTYPE_UINT;
	LENGTH_4_BYTE: typeClassToArgType := Tc2_Utilities.E_ArgType.ARGTYPE_UDINT;
	LENGTH_8_BYTE: typeClassToArgType := Tc2_Utilities.E_ArgType.ARGTYPE_ULARGE;
	ELSE typeClassToArgType := Tc2_Utilities.E_ArgType.ARGTYPE_UNKNOWN;
	END_CASE
ELSE
	typeClassToArgType := Tc2_Utilities.E_ArgType.ARGTYPE_UNKNOWN;
END_CASE
END_METHOD

END_FUNCTION_BLOCK

// ---- AssertionTester/AssertionTests/BitNumberAssertions/classes/ByteAssertionTests.TcPOU
(*

short summary
==================
This class tests all methods of byte assertions
with various combinations of inputs and checks expected 
outputs are satisfied or not

.. <legal notes>

legal notes
=================
| SPDX-FileCopyrightText: © 2022 ekvip automation GmbH <info@ekvip.de>
| SPDX-License-Identifier: Apache-2.0
| For details check: Apache-2.0_

.. _Apache-2.0: https://www.apache.org/licenses/LICENSE-2.0

.. </legal notes>

methods and properties
======================

*)

FUNCTION_BLOCK ByteAssertionTests EXTENDS AbstractAssertorTest
VAR_INPUT
END_VAR
VAR CONSTANT
	(* number of the lsb *)
	FIRST_BIT				:USINT := 0;
	(* number of the msb *)
	LAST_BIT				:USINT := 7;
	(* just the value zero *)
	ZERO					:SINT := 0;
	(* no single bit is set, it's just the value zero *)
	NO_BIT_SET				:BYTE := 16#00;
	(* just the lsb is set, it's just the value one *)
	LSB_ONLY				:BYTE := 16#01;
	(* all bits are set *)
	ALL_BITS_SET			:BYTE := 16#FF;
	(* the msb is set only *)
	MSB_ONLY				:BYTE := 16#80;
	(* prefix to unify the test names *)
	TEST_NAME_PREFIX		:STRING := 'assert.bitNumber.short.';
	(* number how many times the product will be rotated right *)
	NUMBER_OF_RORS			:USINT := 1;
	(* multiplicand for the ``multiplier`` *)
	MULTIPLICAND			:USINT := 16#11;
	(* first of all multipliers the test iterates *)
	FIRST_MULTIPLIER		:USINT := 0;
	(* first of all multipliers the test iterates *)
	LAST_MULTIPLIER			:USINT := 15;
	(* constant for the modulo operator to check if valueToTest is even (lsb is unset) or odd (lsb is set) *)
	DEVISOR_FOR_EVEN_ODD	:USINT := 2;
END_VAR

THIS^.runAndMaskIsEqualToTests();
THIS^.runAndMaskIsNotEqualToTests();
THIS^.runBitXIsEqualToTests();
THIS^.runBitXIsNotEqualToTests();
THIS^.runBitXIsSetTests();
THIS^.runBitXIsUnsetTests();
THIS^.runLsbIsEqualToTests();
THIS^.runLsbIsNotEqualToTests();
THIS^.runLsbIsSetTests();
THIS^.runLsbIsUnsetTests();
THIS^.runMsbIsEqualToTests();
THIS^.runMsbIsNotEqualToTests();
THIS^.runMsbIsSetTests();
THIS^.runMsbIsUnsetTests();
THIS^.runOrMaskIsEqualToTests();
THIS^.runOrMaskIsNotEqualToTests();
THIS^.runValueIsMaxTests();
THIS^.runValueIsMinTests();
THIS^.runValueIsEqualToTests();
THIS^.runValueIsGreaterTests();
THIS^.runValueIsLessThanTests();
THIS^.runValueIsInRangeOfTests();
THIS^.runValueIsNotEqualToTests();
THIS^.runXorMaskIsEqualToTests();
THIS^.runXorMaskIsNotEqualToTests();

(*

short summary
==================
This test method is a helper function to create a unified test name

.. <legal notes>

legal notes
=================
| SPDX-FileCopyrightText: © 2022 ekvip automation GmbH <info@ekvip.de>
| SPDX-License-Identifier: Apache-2.0
| For details check: Apache-2.0_

.. _Apache-2.0: https://www.apache.org/licenses/LICENSE-2.0

.. </legal notes>

parameters
==========

*)

METHOD PROTECTED getTestNameFor :Tc2_System.T_MaxString
VAR_INPUT
	(* name of the method to test, to create a unified test name *)
	nameOfMethodToTest	:Tc2_System.T_MaxString;
END_VAR
getTestNameFor := Tc2_Standard.CONCAT(THIS^.TEST_NAME_PREFIX, nameOfMethodToTest);
END_METHOD

(*

short summary
==================
This test method tests ``assert.bitNumber.short.andMaskIsEqualTo``
method of CNM_AssertionInterfaces library with various inputs

.. <legal notes>

legal notes
=================
| SPDX-FileCopyrightText: © 2022 ekvip automation GmbH <info@ekvip.de>
| SPDX-License-Identifier: Apache-2.0
| For details check: Apache-2.0_

.. _Apache-2.0: https://www.apache.org/licenses/LICENSE-2.0

.. </legal notes>

*)

METHOD runAndMaskIsEqualToTests
VAR
	(* shift to iterate through the bit numbers *)
	shift				:USINT;
	(* mask with the bit iteration *)
	mask				:BYTE;
END_VAR
RETURN (NOT TcUnit.TEST_ORDERED(THIS^.getTestNameFor('AndMaskIsEqualTo')));

FOR shift:= THIS^.FIRST_BIT TO THIS^.LAST_BIT DO
	mask := SHL(THIS^.LSB_ONLY, shift);
	THIS^.testAndMaskIsEqualTo(
		valueToTest := THIS^.ALL_BITS_SET,
		mask  := mask,
		expected := mask
	);
	THIS^.testAndMaskIsEqualTo(
		valueToTest := THIS^.ALL_BITS_SET,
		mask  := mask,
		expected := (NOT mask)
	);
	THIS^.testAndMaskIsEqualTo(
		valueToTest := mask,
		mask  := (NOT mask),
		expected := THIS^.NO_BIT_SET
	);
	THIS^.testAndMaskIsEqualTo(
		valueToTest := mask,
		mask  := (NOT mask),
		expected := (NOT mask)
	);	
	THIS^.testAndMaskIsEqualTo(
		valueToTest := mask,
		mask  := mask,
		expected := mask
	);	
END_FOR

THIS^.testAndMaskIsEqualTo(
	valueToTest := THIS^.NO_BIT_SET,
	mask  := THIS^.NO_BIT_SET,
	expected := THIS^.NO_BIT_SET
);
THIS^.testAndMaskIsEqualTo(
	valueToTest := THIS^.NO_BIT_SET,
	mask  := THIS^.NO_BIT_SET,
	expected := THIS^.LSB_ONLY
);

THIS^.testAndMaskIsEqualTo(
	valueToTest := THIS^.ALL_BITS_SET,
	mask  := THIS^.ALL_BITS_SET,
	expected := THIS^.ALL_BITS_SET
);
THIS^.testAndMaskIsEqualTo(
	valueToTest := THIS^.ALL_BITS_SET,
	mask  := THIS^.ALL_BITS_SET,
	expected := THIS^.NO_BIT_SET
);

TcUnit.TEST_FINISHED();
END_METHOD

(*

short summary
==================
This test method tests ``assert.bitNumber.short.andMaskIsNotEqualTo``
method of CNM_AssertionInterfaces library with various inputs

.. <legal notes>

legal notes
=================
| SPDX-FileCopyrightText: © 2022 ekvip automation GmbH <info@ekvip.de>
| SPDX-License-Identifier: Apache-2.0
| For details check: Apache-2.0_

.. _Apache-2.0: https://www.apache.org/licenses/LICENSE-2.0

.. </legal notes>

*)

METHOD runAndMaskIsNotEqualToTests
VAR
	(* shift to iterate through the bit numbers *)
	shift	:USINT;
	(* mask with the bit iteration *)
	mask	:BYTE;
END_VAR
RETURN (NOT TcUnit.TEST_ORDERED(THIS^.getTestNameFor('AndMaskIsNotEqualTo')));

FOR shift:= THIS^.FIRST_BIT TO THIS^.LAST_BIT DO
	mask := SHL(THIS^.LSB_ONLY, shift);
	THIS^.testAndMaskIsNotEqualTo(
		valueToTest := THIS^.ALL_BITS_SET,
		mask  := mask,
		unexpected := (NOT mask)
	);
	THIS^.testAndMaskIsNotEqualTo(
		valueToTest := THIS^.ALL_BITS_SET,
		mask  := mask,
		unexpected := mask
	);
	THIS^.testAndMaskIsNotEqualTo(
		valueToTest := mask,
		mask  := (NOT mask),
		unexpected := (NOT mask)
	);	
	THIS^.testAndMaskIsNotEqualTo(
		valueToTest := mask,
		mask  := (NOT mask),
		unexpected := THIS^.NO_BIT_SET
	);
	THIS^.testAndMaskIsNotEqualTo(
		valueToTest := mask,
		mask  := mask,
		unexpected := mask
	);	
END_FOR

THIS^.testAndMaskIsNotEqualTo(
	valueToTest := THIS^.NO_BIT_SET,
	mask  := THIS^.NO_BIT_SET,
	unexpected := THIS^.LSB_ONLY
);
THIS^.testAndMaskIsNotEqualTo(
	valueToTest := THIS^.NO_BIT_SET,
	mask  := THIS^.NO_BIT_SET,
	unexpected := THIS^.NO_BIT_SET
);

THIS^.testAndMaskIsNotEqualTo(
	valueToTest := THIS^.ALL_BITS_SET,
	mask  := THIS^.ALL_BITS_SET,
	unexpected := THIS^.NO_BIT_SET
);
THIS^.testAndMaskIsNotEqualTo(
	valueToTest := THIS^.ALL_BITS_SET,
	mask  := THIS^.ALL_BITS_SET,
	unexpected := THIS^.ALL_BITS_SET
);


TcUnit.TEST_FINISHED();
END_METHOD

(*

short summary
==================
This test method tests ``assert.bitNumber.short.bitXIsEqualTo``
method of CNM_AssertionInterfaces library with various inputs

.. <legal notes>

legal notes
=================
| SPDX-FileCopyrightText: © 2022 ekvip automation GmbH <info@ekvip.de>
| SPDX-License-Identifier: Apache-2.0
| For details check: Apache-2.0_

.. _Apache-2.0: https://www.apache.org/licenses/LICENSE-2.0

.. </legal notes>

*)

METHOD runBitXIsEqualToTests
VAR
	(* this is the number of the bit to test *)
	bitNumberToTest	:CNM_AssertionInterfaces.BitNumberByte;
	(* it's just part of the test data *)
	valueToTest		:BYTE;
END_VAR
RETURN (NOT TcUnit.TEST_ORDERED(THIS^.getTestNameFor('bitXIsEqualTo')));

FOR bitNumberToTest := THIS^.FIRST_BIT TO THIS^.LAST_BIT DO

	valueToTest := SHL(THIS^.LSB_ONLY,bitNumberToTest);
	THIS^.testBitXIsEqualTo(
		valueToTest			:=valueToTest,
		bitNumberToCheck	:=bitNumberToTest,
		bitIsSet			:=TRUE
	);
	THIS^.testBitXIsEqualTo(
		valueToTest			:=valueToTest,
		bitNumberToCheck	:=bitNumberToTest,
		bitIsSet			:=FALSE
	);

	valueToTest := (NOT valueToTest);
	THIS^.testBitXIsEqualTo(
		valueToTest			:=valueToTest,
		bitNumberToCheck	:=bitNumberToTest,
		bitIsSet			:=FALSE
	);
	THIS^.testBitXIsEqualTo(
		valueToTest			:=valueToTest,
		bitNumberToCheck	:=bitNumberToTest,
		bitIsSet			:=TRUE
	);	
END_FOR

TcUnit.TEST_FINISHED();
END_METHOD

(*

short summary
==================
This test method tests ``assert.bitNumber.short.bitXIsNotEqualTo``
method of CNM_AssertionInterfaces library with various inputs

.. <legal notes>

legal notes
=================
| SPDX-FileCopyrightText: © 2022 ekvip automation GmbH <info@ekvip.de>
| SPDX-License-Identifier: Apache-2.0
| For details check: Apache-2.0_

.. _Apache-2.0: https://www.apache.org/licenses/LICENSE-2.0

.. </legal notes>

*)

METHOD runBitXIsNotEqualToTests
VAR
	(* this is the number of the bit to test *)
	bitNumberToTest	:CNM_AssertionInterfaces.BitNumberByte;
	(* it's just part of the test data *)
	valueToTest		:BYTE;
END_VAR
RETURN (NOT TcUnit.TEST_ORDERED(THIS^.getTestNameFor('bitXIsNotEqualTo')));

FOR bitNumberToTest := THIS^.FIRST_BIT TO THIS^.LAST_BIT DO
	valueToTest := SHL(THIS^.LSB_ONLY,bitNumberToTest);
	THIS^.testBitXIsNotEqualTo(
		valueToTest			:=valueToTest,
		bitNumberToCheck	:=bitNumberToTest,
		bitIsSet			:=TRUE
	);
	THIS^.testBitXIsNotEqualTo(
		valueToTest			:=valueToTest,
		bitNumberToCheck	:=bitNumberToTest,
		bitIsSet			:=FALSE
	);

	valueToTest := (NOT valueToTest);
	THIS^.testBitXIsNotEqualTo(
		valueToTest			:=valueToTest,
		bitNumberToCheck	:=bitNumberToTest,
		bitIsSet			:=TRUE
	);
	THIS^.testBitXIsNotEqualTo(
		valueToTest			:=valueToTest,
		bitNumberToCheck	:=bitNumberToTest,
		bitIsSet			:=FALSE
	);	
END_FOR

TcUnit.TEST_FINISHED();
END_METHOD

(*

short summary
==================
This test method tests ``assert.bitNumber.short.bitXIsSet`` 
of CNM_AssertionInterfaces library with various inputs

.. <legal notes>

legal notes
=================
| SPDX-FileCopyrightText: © 2022 ekvip automation GmbH <info@ekvip.de>
| SPDX-License-Identifier: Apache-2.0
| For details check: Apache-2.0_

.. _Apache-2.0: https://www.apache.org/licenses/LICENSE-2.0

.. </legal notes>

*)

METHOD runBitXIsSetTests
VAR
	(* this is the number of the bit to test *)
	bitNumberToTest	:CNM_AssertionInterfaces.BitNumberByte;
	(* it's just part of the test data *)
	valueToTest		:BYTE;
END_VAR
RETURN (NOT TcUnit.TEST_ORDERED(THIS^.getTestNameFor('bitXIsSet')));

FOR bitNumberToTest := THIS^.FIRST_BIT TO THIS^.LAST_BIT DO
	valueToTest := SHL(THIS^.LSB_ONLY,bitNumberToTest);
	THIS^.testBitXIsSet(
		valueToTest := valueToTest,
		bitNumberToCheck := bitNumberToTest
	);
	THIS^.testBitXIsSet(
		valueToTest := (NOT valueToTest),
		bitNumberToCheck := bitNumberToTest
	);
	THIS^.testBitXIsSet(
		valueToTest := THIS^.NO_BIT_SET,
		bitNumberToCheck := bitNumberToTest
	);
	THIS^.testBitXIsSet(
		valueToTest := THIS^.ALL_BITS_SET,
		bitNumberToCheck := bitNumberToTest
	);
END_FOR

TcUnit.TEST_FINISHED();
END_METHOD

(*

short summary
==================
This test method tests ``assert.bitNumber.short.bitXIsUnset``
of CNM_AssertionInterfaces library with various inputs

.. <legal notes>

legal notes
=================
| SPDX-FileCopyrightText: © 2022 ekvip automation GmbH <info@ekvip.de>
| SPDX-License-Identifier: Apache-2.0
| For details check: Apache-2.0_

.. _Apache-2.0: https://www.apache.org/licenses/LICENSE-2.0

.. </legal notes>

*)

METHOD runBitXIsUnsetTests
VAR
	(* this is the number of the bit to test *)
	bitNumberToTest	:CNM_AssertionInterfaces.BitNumberByte;
	(* it's just part of the test data *)
	valueToTest		:BYTE;
END_VAR
RETURN (NOT TcUnit.TEST_ORDERED(THIS^.getTestNameFor('bitXIsUnset')));

FOR bitNumberToTest := THIS^.FIRST_BIT TO THIS^.LAST_BIT DO
	valueToTest := SHL(THIS^.LSB_ONLY,bitNumberToTest);
	THIS^.testBitXIsUnset(
		valueToTest := valueToTest,
		bitNumberToCheck := bitNumberToTest
	);
	THIS^.testBitXIsUnset(
		valueToTest := (NOT valueToTest),
		bitNumberToCheck := bitNumberToTest
	);
	THIS^.testBitXIsUnset(
		valueToTest := THIS^.NO_BIT_SET,
		bitNumberToCheck := bitNumberToTest
	);
	THIS^.testBitXIsUnset(
		valueToTest :=THIS^.ALL_BITS_SET,
		bitNumberToCheck := bitNumberToTest
	);
END_FOR

TcUnit.TEST_FINISHED();
END_METHOD

(*

short summary
==================
This test method tests ``assert.bitNumber.short.lsbIsEqualTo``
method of CNM_AssertionInterfaces library with various inputs

.. <legal notes>

legal notes
=================
| SPDX-FileCopyrightText: © 2022 ekvip automation GmbH <info@ekvip.de>
| SPDX-License-Identifier: Apache-2.0
| For details check: Apache-2.0_

.. _Apache-2.0: https://www.apache.org/licenses/LICENSE-2.0

.. </legal notes>

*)

METHOD runLsbIsEqualToTests
VAR
	(* it's just part of the test data *)
	valueToTest	:BYTE;
	(* multiplier to get various bit patterns *)
	multiplier	:USINT;
END_VAR
RETURN (NOT TcUnit.TEST_ORDERED(THIS^.getTestNameFor('lsbIsEqualTo')));

FOR multiplier := THIS^.FIRST_MULTIPLIER TO THIS^.LAST_MULTIPLIER DO
	valueToTest := (THIS^.MULTIPLICAND * multiplier);

	THIS^.testLsbIsEqualTo(
		valueToTest := valueToTest,
		expectedValue := TRUE
	);	
	THIS^.testLsbIsEqualTo(
		valueToTest := valueToTest,
		expectedValue := FALSE
	);

END_FOR

THIS^.testLsbIsEqualTo(
	valueToTest := THIS^.LSB_ONLY,
	expectedValue := TRUE
);	
THIS^.testLsbIsEqualTo(
	valueToTest := THIS^.LSB_ONLY,
	expectedValue := FALSE
);
THIS^.testLsbIsEqualTo(
	valueToTest := THIS^.MSB_ONLY,
	expectedValue := TRUE
);	
THIS^.testLsbIsEqualTo(
	valueToTest := THIS^.MSB_ONLY,
	expectedValue := FALSE
);

TcUnit.TEST_FINISHED();
END_METHOD

(*

short summary
==================
This test method tests ``assert.bitNumber.short.lsbIsNotEqualTo``
method of CNM_AssertionInterfaces library with various inputs

.. <legal notes>

legal notes
=================
| SPDX-FileCopyrightText: © 2022 ekvip automation GmbH <info@ekvip.de>
| SPDX-License-Identifier: Apache-2.0
| For details check: Apache-2.0_

.. _Apache-2.0: https://www.apache.org/licenses/LICENSE-2.0

.. </legal notes>

*)

METHOD runLsbIsNotEqualToTests
VAR
	(* it's just part of the test data *)
	valueToTest	:BYTE;
	(* multiplier to get various bit patterns *)
	multiplier	:USINT;
END_VAR
RETURN (NOT TcUnit.TEST_ORDERED(THIS^.getTestNameFor('lsbIsNotEqualTo')));

FOR multiplier := THIS^.FIRST_MULTIPLIER TO THIS^.LAST_MULTIPLIER DO
	valueToTest := (THIS^.MULTIPLICAND * multiplier);

	THIS^.testLsbIsNotEqualTo(
		valueToTest := valueToTest,
		unexpectedValue := TRUE
	);	
	THIS^.testLsbIsNotEqualTo(
		valueToTest := valueToTest,
		unexpectedValue := FALSE
	);

END_FOR

THIS^.testLsbIsNotEqualTo(
	valueToTest := THIS^.LSB_ONLY,
	unexpectedValue := TRUE
);	
THIS^.testLsbIsNotEqualTo(
	valueToTest := THIS^.LSB_ONLY,
	unexpectedValue := FALSE
);
THIS^.testLsbIsNotEqualTo(
	valueToTest := THIS^.MSB_ONLY,
	unexpectedValue := TRUE
);	
THIS^.testLsbIsNotEqualTo(
	valueToTest := THIS^.MSB_ONLY,
	unexpectedValue := FALSE
);

TcUnit.TEST_FINISHED();
END_METHOD

(*

short summary
==================
This test method tests ``assert.bitNumber.short.lsbIsSet``
of CNM_AssertionInterfaces library with various inputs

.. <legal notes>

legal notes
=================
| SPDX-FileCopyrightText: © 2022 ekvip automation GmbH <info@ekvip.de>
| SPDX-License-Identifier: Apache-2.0
| For details check: Apache-2.0_

.. _Apache-2.0: https://www.apache.org/licenses/LICENSE-2.0

.. </legal notes>

*)

METHOD runLsbIsSetTests
VAR
	(* it's just part of the test data *)
	valueToTest	:BYTE;
	(* multiplier to get various bit patterns *)
	multiplier	:USINT;
END_VAR
RETURN (NOT TcUnit.TEST_ORDERED(THIS^.getTestNameFor('lsbIsSet')));

FOR multiplier := THIS^.FIRST_MULTIPLIER TO THIS^.LAST_MULTIPLIER DO
	valueToTest := (THIS^.MULTIPLICAND * multiplier);
	THIS^.testLsbIsSet(
		valueToTest := valueToTest
	);
END_FOR

THIS^.testLsbIsSet(
	valueToTest := THIS^.MSB_ONLY
);	
THIS^.testLsbIsSet(
	valueToTest := THIS^.MSB_ONLY
);

TcUnit.TEST_FINISHED();
END_METHOD

(*

short summary
==================
This test method tests ``assert.bitNumber.short.lsbIsUnset``
of CNM_AssertionInterfaces library with various inputs

.. <legal notes>

legal notes
=================
| SPDX-FileCopyrightText: © 2022 ekvip automation GmbH <info@ekvip.de>
| SPDX-License-Identifier: Apache-2.0
| For details check: Apache-2.0_

.. _Apache-2.0: https://www.apache.org/licenses/LICENSE-2.0

.. </legal notes>

*)

METHOD runLsbIsUnsetTests
VAR
	(* it's just part of the test data *)
	valueToTest	:BYTE;
	(* multiplier to get various bit patterns *)
	multiplier	:USINT;
END_VAR
RETURN (NOT TcUnit.TEST_ORDERED(THIS^.getTestNameFor('lsbIsUnset')));

FOR multiplier := THIS^.FIRST_MULTIPLIER TO THIS^.LAST_MULTIPLIER DO
	valueToTest := (THIS^.MULTIPLICAND * multiplier);
	THIS^.testLsbIsUnset(
		valueToTest := valueToTest
	);
END_FOR

THIS^.testLsbIsUnset(
	valueToTest := THIS^.LSB_ONLY
);	
THIS^.testLsbIsUnset(
	valueToTest := THIS^.MSB_ONLY
);

TcUnit.TEST_FINISHED();
END_METHOD

(*

short summary
==================
This test method tests ``assert.bitNumber.short.msbIsEqualTo``
method of CNM_AssertionInterfaces library with various inputs

.. <legal notes>

legal notes
=================
| SPDX-FileCopyrightText: © 2022 ekvip automation GmbH <info@ekvip.de>
| SPDX-License-Identifier: Apache-2.0
| For details check: Apache-2.0_

.. _Apache-2.0: https://www.apache.org/licenses/LICENSE-2.0

.. </legal notes>

*)

METHOD runMsbIsEqualToTests
VAR
	(* it's just part of the test data *)
	valueToTest	:BYTE;
	(* multiplier to get various bit patterns *)
	multiplier	:USINT;
END_VAR
VAR CONSTANT
	(* number how many times the product will be rotated right *)
	NUMBER_OF_RORS :USINT := 1;
	(* multiplicand for the ``multiplier`` *)
	MULTIPLICAND :USINT := 17;
	(* first of all multipliers the test iterates *)
	FIRST_MULTIPLIER :USINT := 0;
	(* first of all multipliers the test iterates *)
	LAST_MULTIPLIER :USINT := 15;
END_VAR
RETURN (NOT TcUnit.TEST_ORDERED(THIS^.getTestNameFor('msbIsEqualTo')));

FOR multiplier := THIS^.FIRST_MULTIPLIER TO THIS^.LAST_MULTIPLIER DO
	valueToTest := ROR(THIS^.MULTIPLICAND * multiplier, THIS^.NUMBER_OF_RORS);

	THIS^.testMsbIsEqualTo(
		valueToTest := valueToTest,
		expectedValue := TRUE
	);	
	THIS^.testMsbIsEqualTo(
		valueToTest := valueToTest,
		expectedValue := FALSE
	);
END_FOR

THIS^.testMsbIsEqualTo(
	valueToTest := THIS^.LSB_ONLY,
	expectedValue := TRUE
);	
THIS^.testMsbIsEqualTo(
	valueToTest := THIS^.LSB_ONLY,
	expectedValue := FALSE
);
THIS^.testMsbIsEqualTo(
	valueToTest := THIS^.MSB_ONLY,
	expectedValue := TRUE
);	
THIS^.testMsbIsEqualTo(
	valueToTest := THIS^.MSB_ONLY,
	expectedValue := FALSE
);

TcUnit.TEST_FINISHED();
END_METHOD

(*

short summary
==================
This test method tests ``assert.bitNumber.short.msbIsNotEqualTo``
method of CNM_AssertionInterfaces library with various inputs

.. <legal notes>

legal notes
=================
| SPDX-FileCopyrightText: © 2022 ekvip automation GmbH <info@ekvip.de>
| SPDX-License-Identifier: Apache-2.0
| For details check: Apache-2.0_

.. _Apache-2.0: https://www.apache.org/licenses/LICENSE-2.0

.. </legal notes>

*)

METHOD runMsbIsNotEqualToTests
VAR
	(* it's just part of the test data *)
	valueToTest	:BYTE;
	(* multiplier to get various bit patterns *)
	multiplier	:USINT;
END_VAR
RETURN (NOT TcUnit.TEST_ORDERED(THIS^.getTestNameFor('msbIsNotEqualTo')));

FOR multiplier := THIS^.FIRST_MULTIPLIER TO THIS^.LAST_MULTIPLIER DO
	valueToTest := ROR(THIS^.MULTIPLICAND * multiplier, THIS^.NUMBER_OF_RORS);
	THIS^.testMsbIsNotEqualTo(
		valueToTest := valueToTest,
		unexpectedValue := TRUE
	);	
	THIS^.testMsbIsNotEqualTo(
		valueToTest := valueToTest,
		unexpectedValue := FALSE
	);
END_FOR

THIS^.testMsbIsNotEqualTo(
	valueToTest := THIS^.LSB_ONLY,
	unexpectedValue := TRUE
);	
THIS^.testMsbIsNotEqualTo(
	valueToTest := THIS^.LSB_ONLY,
	unexpectedValue := FALSE
);
THIS^.testMsbIsNotEqualTo(
	valueToTest := THIS^.MSB_ONLY,
	unexpectedValue := TRUE
);	
THIS^.testMsbIsNotEqualTo(
	valueToTest := THIS^.MSB_ONLY,
	unexpectedValue := FALSE
);

TcUnit.TEST_FINISHED();
END_METHOD

(*

short summary
==================
This test method tests ``assert.bitNumber.short.msbIsSet``
of CNM_AssertionInterfaces library with various inputs

.. <legal notes>

legal notes
=================
| SPDX-FileCopyrightText: © 2022 ekvip automation GmbH <info@ekvip.de>
| SPDX-License-Identifier: Apache-2.0
| For details check: Apache-2.0_

.. _Apache-2.0: https://www.apache.org/licenses/LICENSE-2.0

.. </legal notes>

*)

METHOD runMsbIsSetTests
VAR
	(* it's just part of the test data *)
	valueToTest	:BYTE;
	(* multiplier to get various bit patterns *)
	multiplier	:USINT;
END_VAR
RETURN (NOT TcUnit.TEST_ORDERED(THIS^.getTestNameFor('msbIsUnset')));

FOR multiplier := THIS^.FIRST_MULTIPLIER TO THIS^.LAST_MULTIPLIER DO
	valueToTest := ROR(THIS^.MULTIPLICAND * multiplier, THIS^.NUMBER_OF_RORS);
	THIS^.testMsbIsSet(
		valueToTest := valueToTest
	);
END_FOR

THIS^.testMsbIsSet(
	valueToTest := THIS^.LSB_ONLY
);	
THIS^.testMsbIsSet(
	valueToTest := THIS^.MSB_ONLY
);

TcUnit.TEST_FINISHED();
END_METHOD

(*

short summary
==================
This test method tests ``assert.bitNumber.short.msbIsUnset``
of CNM_AssertionInterfaces library with various inputs

.. <legal notes>

legal notes
=================
| SPDX-FileCopyrightText: © 2022 ekvip automation GmbH <info@ekvip.de>
| SPDX-License-Identifier: Apache-2.0
| For details check: Apache-2.0_

.. _Apache-2.0: https://www.apache.org/licenses/LICENSE-2.0

.. </legal notes>

*)

METHOD runMsbIsUnsetTests
VAR
	(* it's just part of the test data *)
	valueToTest	:BYTE;
	(* multiplier to get various bit patterns *)
	multiplier	:USINT;
END_VAR
RETURN (NOT TcUnit.TEST_ORDERED(THIS^.getTestNameFor('msbIsSet')));

FOR multiplier := THIS^.FIRST_MULTIPLIER TO THIS^.LAST_MULTIPLIER DO
	valueToTest := ROR(THIS^.MULTIPLICAND * multiplier, THIS^.NUMBER_OF_RORS);
	THIS^.testMsbIsSet(
		valueToTest := valueToTest
	);
END_FOR

THIS^.testMsbIsSet(
	valueToTest := THIS^.LSB_ONLY
);	
THIS^.testMsbIsSet(
	valueToTest := THIS^.MSB_ONLY
);

TcUnit.TEST_FINISHED();
END_METHOD

(*

short summary
==================
This test method tests ``assert.bitNumber.short.orMaskIsEqualTo``
method of CNM_AssertionInterfaces library with various inputs

.. <legal notes>

legal notes
=================
| SPDX-FileCopyrightText: © 2022 ekvip automation GmbH <info@ekvip.de>
| SPDX-License-Identifier: Apache-2.0
| For details check: Apache-2.0_

.. _Apache-2.0: https://www.apache.org/licenses/LICENSE-2.0

.. </legal notes>

*)

METHOD runOrMaskIsEqualToTests
VAR
	(* shift to iterate through the bit numbers *)
	shift				:USINT;
	(* it's just part of the test data *)
	valueToTest		:BYTE;
	(* mask with the bit iteration *)
	mask				:BYTE;
END_VAR
RETURN (NOT TcUnit.TEST_ORDERED(THIS^.getTestNameFor('orMaskIsEqualTo')));

FOR shift:= THIS^.FIRST_BIT TO THIS^.LAST_BIT DO
	mask := SHL(THIS^.LSB_ONLY, shift);
	valueToTest := SHR(THIS^.MSB_ONLY, shift);
	THIS^.testOrMaskIsEqualTo(
		valueToTest := valueToTest,
		mask  := mask,
		expected := (mask OR valueToTest)
	);
	THIS^.testOrMaskIsEqualTo(
		valueToTest := valueToTest,
		mask  := mask,
		expected := (NOT (mask OR valueToTest))
	);
	THIS^.testAndMaskIsEqualTo(
		valueToTest := mask,
		mask  := (NOT mask),
		expected := THIS^.NO_BIT_SET
	);
	THIS^.testAndMaskIsEqualTo(
		valueToTest := mask,
		mask  := (NOT mask),
		expected := THIS^.ALL_BITS_SET
	);	
END_FOR

THIS^.testAndMaskIsEqualTo(
	valueToTest := THIS^.NO_BIT_SET,
	mask  := THIS^.NO_BIT_SET,
	expected := THIS^.NO_BIT_SET
);
THIS^.testAndMaskIsEqualTo(
	valueToTest := THIS^.NO_BIT_SET,
	mask  := THIS^.NO_BIT_SET,
	expected := THIS^.ALL_BITS_SET
);	

THIS^.testAndMaskIsEqualTo(
	valueToTest := THIS^.ALL_BITS_SET,
	mask  := THIS^.ALL_BITS_SET,
	expected := THIS^.ALL_BITS_SET
);
THIS^.testAndMaskIsEqualTo(
	valueToTest := THIS^.ALL_BITS_SET,
	mask  := THIS^.ALL_BITS_SET,
	expected := THIS^.NO_BIT_SET
);	

TcUnit.TEST_FINISHED();
END_METHOD

(*

short summary
==================
This test method tests ``assert.bitNumber.short.orMaskIsNotEqualTo``
method of CNM_AssertionInterfaces library with various inputs

.. <legal notes>

legal notes
=================
| SPDX-FileCopyrightText: © 2022 ekvip automation GmbH <info@ekvip.de>
| SPDX-License-Identifier: Apache-2.0
| For details check: Apache-2.0_

.. _Apache-2.0: https://www.apache.org/licenses/LICENSE-2.0

.. </legal notes>

*)

METHOD runOrMaskIsNotEqualToTests
VAR
	(* shift to iterate through the bit numbers *)
	shift				:USINT;
	(* it's just part of the test data *)
	valueToTest		:BYTE;
	(* mask with the bit iteration *)
	mask				:BYTE;
END_VAR
RETURN (NOT TcUnit.TEST_ORDERED(THIS^.getTestNameFor('orMaskIsNotEqualTo')));

FOR shift:= THIS^.FIRST_BIT TO THIS^.LAST_BIT DO
	mask := SHL(THIS^.LSB_ONLY, shift);
	valueToTest := SHR(THIS^.MSB_ONLY, shift);
	THIS^.testOrMaskIsNotEqualTo(
		valueToTest := valueToTest,
		mask  := mask,
		unexpected := (mask OR valueToTest)
	);
	THIS^.testOrMaskIsNotEqualTo(
		valueToTest := valueToTest,
		mask  := mask,
		unexpected := (NOT (mask OR valueToTest))
	);
	THIS^.testOrMaskIsNotEqualTo(
		valueToTest := mask,
		mask  := (NOT mask),
		unexpected := THIS^.NO_BIT_SET
	);
	THIS^.testOrMaskIsNotEqualTo(
		valueToTest := mask,
		mask  := (NOT mask),
		unexpected := THIS^.ALL_BITS_SET
	);	
END_FOR

THIS^.testOrMaskIsNotEqualTo(
	valueToTest := THIS^.NO_BIT_SET,
	mask  := THIS^.NO_BIT_SET,
	unexpected := THIS^.NO_BIT_SET
);
THIS^.testOrMaskIsNotEqualTo(
	valueToTest := THIS^.NO_BIT_SET,
	mask  := THIS^.NO_BIT_SET,
	unexpected := THIS^.ALL_BITS_SET
);	

THIS^.testOrMaskIsNotEqualTo(
	valueToTest := THIS^.ALL_BITS_SET,
	mask  := THIS^.ALL_BITS_SET,
	unexpected := THIS^.ALL_BITS_SET
);
THIS^.testOrMaskIsNotEqualTo(
	valueToTest := THIS^.ALL_BITS_SET,
	mask  := THIS^.ALL_BITS_SET,
	unexpected := THIS^.NO_BIT_SET
);	

TcUnit.TEST_FINISHED();
END_METHOD

(*

short summary
==================
This test method tests ``assert.bitNumber.short.valueIsEqualTo``
method of CNM_AssertionInterfaces library with various inputs

.. <legal notes>

legal notes
=================
| SPDX-FileCopyrightText: © 2022 ekvip automation GmbH <info@ekvip.de>
| SPDX-License-Identifier: Apache-2.0
| For details check: Apache-2.0_

.. _Apache-2.0: https://www.apache.org/licenses/LICENSE-2.0

.. </legal notes>

*)

METHOD runValueIsEqualToTests
RETURN (NOT TcUnit.TEST_ORDERED(THIS^.getTestNameFor('valueIsEqualTo')));

THIS^.testValueIsEqualTo(
	valueToTest := THIS^.NO_BIT_SET,
	expected := THIS^.ALL_BITS_SET
);
THIS^.testValueIsEqualTo(
	valueToTest := THIS^.NO_BIT_SET,
	expected := THIS^.NO_BIT_SET
);
THIS^.testValueIsEqualTo(
	valueToTest := THIS^.ALL_BITS_SET,
	expected := THIS^.ALL_BITS_SET
);
THIS^.testValueIsEqualTo(
	valueToTest := THIS^.ALL_BITS_SET,
	expected := THIS^.NO_BIT_SET
);
THIS^.testValueIsEqualTo(
	valueToTest := THIS^.LSB_ONLY,
	expected := THIS^.LSB_ONLY
);
THIS^.testValueIsEqualTo(
	valueToTest := THIS^.LSB_ONLY,
	expected := THIS^.MSB_ONLY
);
THIS^.testValueIsEqualTo(
	valueToTest := THIS^.MSB_ONLY,
	expected := THIS^.MSB_ONLY
);
THIS^.testValueIsEqualTo(
	valueToTest := THIS^.MSB_ONLY,
	expected := THIS^.LSB_ONLY
);

TcUnit.TEST_FINISHED();
END_METHOD

(*

short summary
==================
This test method tests ``assert.bitNumber.short.valueIsGreaterThan``
method of CNM_AssertionInterfaces library with various inputs

.. <legal notes>

legal notes
=================
| SPDX-FileCopyrightText: © 2022 ekvip automation GmbH <info@ekvip.de>
| SPDX-License-Identifier: Apache-2.0
| For details check: Apache-2.0_

.. _Apache-2.0: https://www.apache.org/licenses/LICENSE-2.0

.. </legal notes>

*)

METHOD runValueIsGreaterTests
RETURN (NOT TcUnit.TEST_ORDERED(THIS^.getTestNameFor('valueIsGreaterThan')));

THIS^.testValueIsGreater(
	valueToTest := THIS^.NO_BIT_SET,
	less := THIS^.ALL_BITS_SET
);
THIS^.testValueIsGreater(
	valueToTest := THIS^.NO_BIT_SET,
	less := THIS^.NO_BIT_SET
);
THIS^.testValueIsGreater(
	valueToTest := THIS^.ALL_BITS_SET,
	less := THIS^.ALL_BITS_SET
);
THIS^.testValueIsGreater(
	valueToTest := THIS^.ALL_BITS_SET,
	less := THIS^.NO_BIT_SET
);
THIS^.testValueIsGreater(
	valueToTest := THIS^.LSB_ONLY,
	less := THIS^.LSB_ONLY
);
THIS^.testValueIsGreater(
	valueToTest := THIS^.LSB_ONLY,
	less := THIS^.NO_BIT_SET
);
THIS^.testValueIsGreater(
	valueToTest := THIS^.LSB_ONLY,
	less := (THIS^.LSB_ONLY+THIS^.LSB_ONLY)
);
THIS^.testValueIsGreater(
	valueToTest := THIS^.MSB_ONLY,
	less := THIS^.MSB_ONLY
);
THIS^.testValueIsGreater(
	valueToTest := THIS^.MSB_ONLY,
	less := (NOT THIS^.MSB_ONLY)
);
THIS^.testValueIsGreater(
	valueToTest := THIS^.MSB_ONLY,
	less := THIS^.ALL_BITS_SET
);

TcUnit.TEST_FINISHED();
END_METHOD

(*

short summary
==================
This test method tests ``assert.bitNumber.short.valueIsInRangeOf``
method of CNM_AssertionInterfaces library with various inputs

.. <legal notes>

legal notes
=================
| SPDX-FileCopyrightText: © 2022 ekvip automation GmbH <info@ekvip.de>
| SPDX-License-Identifier: Apache-2.0
| For details check: Apache-2.0_

.. _Apache-2.0: https://www.apache.org/licenses/LICENSE-2.0

.. </legal notes>

*)

METHOD runValueIsInRangeOfTests
RETURN (NOT TcUnit.TEST_ORDERED(THIS^.getTestNameFor('valueIsInRangeOf')));

THIS^.testValueIsInRangeOf(
	lower := THIS^.NO_BIT_SET,
	valueToTest := THIS^.LSB_ONLY,
	upper := THIS^.ALL_BITS_SET
);
THIS^.testValueIsInRangeOf(
	lower := THIS^.NO_BIT_SET,
	valueToTest := THIS^.NO_BIT_SET,
	upper := THIS^.NO_BIT_SET
);
THIS^.testValueIsInRangeOf(
	lower := THIS^.ALL_BITS_SET,
	valueToTest := THIS^.ALL_BITS_SET,
	upper := THIS^.ALL_BITS_SET
);
THIS^.testValueIsInRangeOf(
	lower := THIS^.ALL_BITS_SET,
	valueToTest := THIS^.LSB_ONLY,
	upper := THIS^.NO_BIT_SET
);
THIS^.testValueIsInRangeOf(
	lower := THIS^.ALL_BITS_SET,
	valueToTest := THIS^.NO_BIT_SET,
	upper := THIS^.NO_BIT_SET
);

TEST_FINISHED();
END_METHOD

(*

short summary
==================
This test method tests ``assert.bitNumber.short.valueIsLessThan``
method of CNM_AssertionInterfaces library with various inputs

.. <legal notes>

legal notes
=================
| SPDX-FileCopyrightText: © 2022 ekvip automation GmbH <info@ekvip.de>
| SPDX-License-Identifier: Apache-2.0
| For details check: Apache-2.0_

.. _Apache-2.0: https://www.apache.org/licenses/LICENSE-2.0

.. </legal notes>

*)

METHOD runValueIsLessThanTests
RETURN (NOT TcUnit.TEST_ORDERED(THIS^.getTestNameFor('valueIsLessThan')));

THIS^.testValueIsLessThan(
	valueToTest := THIS^.NO_BIT_SET,
	greater := THIS^.ALL_BITS_SET
);
THIS^.testValueIsLessThan(
	valueToTest := THIS^.NO_BIT_SET,
	greater := THIS^.NO_BIT_SET
);
THIS^.testValueIsLessThan(
	valueToTest := THIS^.ALL_BITS_SET,
	greater := THIS^.ALL_BITS_SET
);
THIS^.testValueIsLessThan(
	valueToTest := THIS^.ALL_BITS_SET,
	greater := THIS^.NO_BIT_SET
);
THIS^.testValueIsLessThan(
	valueToTest := THIS^.LSB_ONLY,
	greater := THIS^.LSB_ONLY
);
THIS^.testValueIsLessThan(
	valueToTest := THIS^.LSB_ONLY,
	greater := THIS^.NO_BIT_SET
);
THIS^.testValueIsLessThan(
	valueToTest := THIS^.MSB_ONLY,
	greater := (THIS^.MSB_ONLY+THIS^.LSB_ONLY)
);
THIS^.testValueIsLessThan(
	valueToTest := THIS^.MSB_ONLY,
	greater := THIS^.MSB_ONLY
);
THIS^.testValueIsLessThan(
	valueToTest := THIS^.MSB_ONLY,
	greater := (NOT THIS^.MSB_ONLY)
);
THIS^.testValueIsLessThan(
	valueToTest := THIS^.MSB_ONLY,
	greater := THIS^.ALL_BITS_SET
);

TcUnit.TEST_FINISHED();
END_METHOD

(*

short summary
==================
This test method tests ``assert.bitNumber.short.valueIsMax``
method of CNM_AssertionInterfaces library with various inputs

.. <legal notes>

legal notes
=================
| SPDX-FileCopyrightText: © 2022 ekvip automation GmbH <info@ekvip.de>
| SPDX-License-Identifier: Apache-2.0
| For details check: Apache-2.0_

.. _Apache-2.0: https://www.apache.org/licenses/LICENSE-2.0

.. </legal notes>

*)

METHOD runValueIsMaxTests
RETURN (NOT TcUnit.TEST_ORDERED(THIS^.getTestNameFor('valueIsMax')));

THIS^.testValueIsMax(
	valueToTest := THIS^.NO_BIT_SET,
	maximum := THIS^.LSB_ONLY
);
THIS^.testValueIsMax(
	valueToTest := THIS^.LSB_ONLY,
	maximum := THIS^.NO_BIT_SET
);
THIS^.testValueIsMax(
	valueToTest := THIS^.NO_BIT_SET,
	maximum := THIS^.NO_BIT_SET
);
THIS^.testValueIsMax(
	valueToTest := THIS^.ALL_BITS_SET,
	maximum := ALL_BITS_SET
);
THIS^.testValueIsMax(
	valueToTest := (THIS^.ALL_BITS_SET-THIS^.LSB_ONLY),
	maximum := THIS^.ALL_BITS_SET
);
THIS^.testValueIsMax(
	valueToTest := THIS^.ALL_BITS_SET,
	maximum := (THIS^.ALL_BITS_SET-THIS^.LSB_ONLY)
);
THIS^.testValueIsMax(
	valueToTest := THIS^.MSB_ONLY,
	maximum := (THIS^.MSB_ONLY+THIS^.LSB_ONLY)
);
THIS^.testValueIsMax(
	valueToTest := (THIS^.MSB_ONLY+THIS^.LSB_ONLY),
	maximum := THIS^.MSB_ONLY
);
THIS^.testValueIsMax(
	valueToTest := THIS^.MSB_ONLY,
	maximum := (NOT THIS^.MSB_ONLY)
);
THIS^.testValueIsMax(
	valueToTest := (NOT THIS^.MSB_ONLY),
	maximum := THIS^.MSB_ONLY
);
THIS^.testValueIsMax(
	valueToTest := THIS^.MSB_ONLY,
	maximum := THIS^.MSB_ONLY
);

TcUnit.TEST_FINISHED();
END_METHOD

(*

short summary
==================
This test method tests ``assert.bitNumber.short.valueIsMin``
method of CNM_AssertionInterfaces library with various inputs

.. <legal notes>

legal notes
=================
| SPDX-FileCopyrightText: © 2022 ekvip automation GmbH <info@ekvip.de>
| SPDX-License-Identifier: Apache-2.0
| For details check: Apache-2.0_

.. _Apache-2.0: https://www.apache.org/licenses/LICENSE-2.0

.. </legal notes>

*)

METHOD runValueIsMinTests
RETURN (NOT TcUnit.TEST_ORDERED(THIS^.getTestNameFor('valueIsMin')));

THIS^.testValueIsMin(
	valueToTest := THIS^.NO_BIT_SET,
	minimum := THIS^.LSB_ONLY
);
THIS^.testValueIsMin(
	valueToTest := THIS^.LSB_ONLY,
	minimum := THIS^.NO_BIT_SET
);
THIS^.testValueIsMin(
	valueToTest := THIS^.NO_BIT_SET,
	minimum := THIS^.NO_BIT_SET
);
THIS^.testValueIsMin(
	valueToTest := THIS^.ALL_BITS_SET,
	minimum := ALL_BITS_SET
);
THIS^.testValueIsMin(
	valueToTest := (THIS^.ALL_BITS_SET-THIS^.LSB_ONLY),
	minimum := THIS^.ALL_BITS_SET
);
THIS^.testValueIsMin(
	valueToTest := THIS^.ALL_BITS_SET,
	minimum := (THIS^.ALL_BITS_SET-THIS^.LSB_ONLY)
);
THIS^.testValueIsMin(
	valueToTest := THIS^.MSB_ONLY,
	minimum := (THIS^.MSB_ONLY+THIS^.LSB_ONLY)
);
THIS^.testValueIsMin(
	valueToTest := (THIS^.MSB_ONLY+THIS^.LSB_ONLY),
	minimum := THIS^.MSB_ONLY
);
THIS^.testValueIsMin(
	valueToTest := THIS^.MSB_ONLY,
	minimum := (NOT THIS^.MSB_ONLY)
);
THIS^.testValueIsMin(
	valueToTest := (NOT THIS^.MSB_ONLY),
	minimum := THIS^.MSB_ONLY
);
THIS^.testValueIsMin(
	valueToTest := THIS^.MSB_ONLY,
	minimum := THIS^.MSB_ONLY
);

TcUnit.TEST_FINISHED();
END_METHOD

(*

short summary
==================
This test method tests ``assert.bitNumber.short.valueIsNotEqualTo``
method of CNM_AssertionInterfaces library with various inputs

.. <legal notes>

legal notes
=================
| SPDX-FileCopyrightText: © 2022 ekvip automation GmbH <info@ekvip.de>
| SPDX-License-Identifier: Apache-2.0
| For details check: Apache-2.0_

.. _Apache-2.0: https://www.apache.org/licenses/LICENSE-2.0

.. </legal notes>

*)

METHOD runValueIsNotEqualToTests
RETURN (NOT TcUnit.TEST_ORDERED(THIS^.getTestNameFor('valueIsNotEqualTo')));

THIS^.testValueIsNotEqualTo(
	valueToTest := THIS^.NO_BIT_SET,
	unexpected := THIS^.ALL_BITS_SET
);
THIS^.testValueIsNotEqualTo(
	valueToTest := THIS^.NO_BIT_SET,
	unexpected := THIS^.NO_BIT_SET
);
THIS^.testValueIsNotEqualTo(
	valueToTest := THIS^.ALL_BITS_SET,
	unexpected := THIS^.ALL_BITS_SET
);
THIS^.testValueIsNotEqualTo(
	valueToTest := THIS^.ALL_BITS_SET,
	unexpected := THIS^.NO_BIT_SET
);
THIS^.testValueIsNotEqualTo(
	valueToTest := THIS^.LSB_ONLY,
	unexpected := THIS^.LSB_ONLY
);
THIS^.testValueIsNotEqualTo(
	valueToTest := THIS^.LSB_ONLY,
	unexpected := THIS^.MSB_ONLY
);
THIS^.testValueIsNotEqualTo(
	valueToTest := THIS^.MSB_ONLY,
	unexpected := THIS^.MSB_ONLY
);
THIS^.testValueIsNotEqualTo(
	valueToTest := THIS^.MSB_ONLY,
	unexpected := THIS^.LSB_ONLY
);

TcUnit.TEST_FINISHED();
END_METHOD

(*

short summary
==================
This test method tests ``assert.bitNumber.short.xorMaskIsEqualTo``
method of CNM_AssertionInterfaces library with various inputs

.. <legal notes>

legal notes
=================
| SPDX-FileCopyrightText: © 2022 ekvip automation GmbH <info@ekvip.de>
| SPDX-License-Identifier: Apache-2.0
| For details check: Apache-2.0_

.. _Apache-2.0: https://www.apache.org/licenses/LICENSE-2.0

.. </legal notes>

*)

METHOD runXorMaskIsEqualToTests
VAR
	(* shift to iterate through the bit numbers *)
	shift				:USINT;
	(* it's just part of the test data *)
	valueToTest		:BYTE;
	(* mask with the bit iteration *)
	mask				:BYTE;
END_VAR
RETURN (NOT TcUnit.TEST_ORDERED(THIS^.getTestNameFor('xorMaskIsEqualTo')));

FOR shift:= THIS^.FIRST_BIT TO THIS^.LAST_BIT DO
	mask := SHL(THIS^.LSB_ONLY, shift);
	valueToTest := (NOT mask);
	THIS^.testOrMaskIsEqualTo(
		valueToTest := valueToTest,
		mask  := mask,
		expected := THIS^.ALL_BITS_SET
	);
	THIS^.testOrMaskIsEqualTo(
		valueToTest := valueToTest,
		mask  := mask,
		expected := THIS^.NO_BIT_SET
	);
	THIS^.testAndMaskIsEqualTo(
		valueToTest := mask,
		mask  := mask,
		expected := THIS^.NO_BIT_SET
	);
	THIS^.testAndMaskIsEqualTo(
		valueToTest := mask,
		mask  := mask,
		expected := mask
	);	
END_FOR

THIS^.testAndMaskIsEqualTo(
	valueToTest := THIS^.NO_BIT_SET,
	mask  := THIS^.NO_BIT_SET,
	expected := THIS^.NO_BIT_SET
);
THIS^.testAndMaskIsEqualTo(
	valueToTest := THIS^.NO_BIT_SET,
	mask  := THIS^.NO_BIT_SET,
	expected := THIS^.ALL_BITS_SET
);	

THIS^.testAndMaskIsEqualTo(
	valueToTest := THIS^.ALL_BITS_SET,
	mask  := THIS^.ALL_BITS_SET,
	expected := THIS^.ALL_BITS_SET
);
THIS^.testAndMaskIsEqualTo(
	valueToTest := THIS^.ALL_BITS_SET,
	mask  := THIS^.ALL_BITS_SET,
	expected := THIS^.NO_BIT_SET
);	

TcUnit.TEST_FINISHED();
END_METHOD

(*

short summary
==================
This test method tests ``assert.bitNumber.short.xorMaskIsNotEqualTo``
method of CNM_AssertionInterfaces library with various inputs

.. <legal notes>

legal notes
=================
| SPDX-FileCopyrightText: © 2022 ekvip automation GmbH <info@ekvip.de>
| SPDX-License-Identifier: Apache-2.0
| For details check: Apache-2.0_

.. _Apache-2.0: https://www.apache.org/licenses/LICENSE-2.0

.. </legal notes>

*)

METHOD runXorMaskIsNotEqualToTests
VAR
	(* shift to iterate through the bit numbers *)
	shift				:USINT;
	(* it's just part of the test data *)
	valueToTest			:BYTE;
	(* mask with the bit iteration *)
	mask				:BYTE;
END_VAR
RETURN (NOT TcUnit.TEST_ORDERED(THIS^.getTestNameFor('xorMaskIsNotEqualTo')));

FOR shift:= THIS^.FIRST_BIT TO THIS^.LAST_BIT DO
	mask := SHL(THIS^.LSB_ONLY, shift);
	valueToTest := (NOT mask);
	THIS^.testXorMaskIsNotEqualTo(
		valueToTest := valueToTest,
		mask  := mask,
		unexpected := THIS^.ALL_BITS_SET
	);
	THIS^.testXorMaskIsNotEqualTo(
		valueToTest := valueToTest,
		mask  := mask,
		unexpected := THIS^.NO_BIT_SET
	);
	THIS^.testXorMaskIsNotEqualTo(
		valueToTest := mask,
		mask  := mask,
		unexpected := THIS^.NO_BIT_SET
	);
	THIS^.testXorMaskIsNotEqualTo(
		valueToTest := mask,
		mask  := mask,
		unexpected := mask
	);	
END_FOR

THIS^.testXorMaskIsNotEqualTo(
	valueToTest := THIS^.NO_BIT_SET,
	mask  := THIS^.NO_BIT_SET,
	unexpected := THIS^.NO_BIT_SET
);
THIS^.testXorMaskIsNotEqualTo(
	valueToTest := THIS^.NO_BIT_SET,
	mask  := THIS^.NO_BIT_SET,
	unexpected := THIS^.ALL_BITS_SET
);	

THIS^.testXorMaskIsNotEqualTo(
	valueToTest := THIS^.ALL_BITS_SET,
	mask  := THIS^.ALL_BITS_SET,
	unexpected := THIS^.ALL_BITS_SET
);
THIS^.testXorMaskIsNotEqualTo(
	valueToTest := THIS^.ALL_BITS_SET,
	mask  := THIS^.ALL_BITS_SET,
	unexpected := THIS^.NO_BIT_SET
);	

THIS^.testXorMaskIsNotEqualTo(
	valueToTest := THIS^.ALL_BITS_SET,
	mask  := THIS^.NO_BIT_SET,
	unexpected := THIS^.ALL_BITS_SET
);
THIS^.testXorMaskIsNotEqualTo(
	valueToTest := THIS^.ALL_BITS_SET,
	mask  := THIS^.NO_BIT_SET,
	unexpected := THIS^.NO_BIT_SET
);

TcUnit.TEST_FINISHED();
END_METHOD

(*

short summary
==================
This test method tests ``assert.bitNumber.short.andMaskIsEqualTo``
method of CNM_AssertionInterfaces library, 
it provides the possibility to handover test data via parameter 


.. <legal notes>

legal notes
=================
| SPDX-FileCopyrightText: © 2022 ekvip automation GmbH <info@ekvip.de>
| SPDX-License-Identifier: Apache-2.0
| For details check: Apache-2.0_

.. _Apache-2.0: https://www.apache.org/licenses/LICENSE-2.0

.. </legal notes>

parameters
==========

*)

METHOD testAndMaskIsEqualTo 
VAR_INPUT
	(* for the test it's the parameter ``currentValue`` *)
	valueToTest	:BYTE;
	(* it's the mask for the currentValue *)
	mask		:BYTE;
	(* for the test it's the parameter ``expectedValue`` *)
	expected	:BYTE;
END_VAR
VAR
	(* just the expectation if the assertion to test must be worng or true *)
	assertionIsWrong		:BOOL;
	(* result of the bit operation to determine the value of ``assertionIsWrong`` *)
	result					:BYTE;
	(* contains the format string for the test message *)
	message					:Tc2_System.T_MaxString;
	(* TwinCAT printf with the test message *)
	messageStringBuilder	:Tc2_Utilities.FB_FormatString;
END_VAR
THIS^.assertorContainer.resetAssertor();

result := (valueToTest AND mask);
assertionIsWrong := (result <> expected);
message := SEL(
	assertionIsWrong,
	'currentValue: 16#%.2X AND mask: 16#%.2X is 16#%.2X expectedValue: 16#%.2X assertion must be TRUE', 
	'currentValue: 16#%.2X AND mask: 16#%.2X is 16#%.2X expectedValue: 16#%.2X assertion must be FALSE'
);
messageStringBuilder(
	sFormat := message,
	arg1 := THIS^.AnyToArg(valueToTest),
	arg2 := THIS^.AnyToArg(mask),
	arg3 := THIS^.AnyToArg(result),
	arg4 := THIS^.AnyToArg(expected)
);

THIS^.assertorContainer.assertor.assert.bitNumber.short.andMaskIsEqualTo(
	currentValue	:= valueToTest,
	mask 			:= mask,
	expectedValue	:= expected,
	message			:= ''
);

THIS^.AssertEquals_BOOL(
	Expected 	:= assertionIsWrong,
	Actual 		:= THIS^.assertorContainer.wasAssertionWrong,
	Message 	:= messageStringBuilder.sOut
);
END_METHOD

(*

short summary
==================
This test method tests ``assert.bitNumber.short.andMaskIsNotEqualTo``
method of CNM_AssertionInterfaces library, 
it provides the possibility to handover test data via parameter 


.. <legal notes>

legal notes
=================
| SPDX-FileCopyrightText: © 2022 ekvip automation GmbH <info@ekvip.de>
| SPDX-License-Identifier: Apache-2.0
| For details check: Apache-2.0_

.. _Apache-2.0: https://www.apache.org/licenses/LICENSE-2.0

.. </legal notes>

parameters
==========

*)

METHOD testAndMaskIsNotEqualTo 
VAR_INPUT
	(* for the test it's the parameter ``currentValue`` *)
	valueToTest	:BYTE;
	(* it's the mask for the currentValue *)
	mask		:BYTE;
	(* for the test it's the parameter ``unexpectedValue`` *)
	unexpected	:BYTE;
END_VAR
VAR
	(* just the expectation if the assertion to test must be worng or true *)
	assertionIsWrong		:BOOL;
	(* result of the bit operation to determine the value of ``assertionIsWrong`` *)
	result					:BYTE;
	(* contains the format string for the test message *)
	message					:Tc2_System.T_MaxString;
	(* TwinCAT printf with the test message *)
	messageStringBuilder	:Tc2_Utilities.FB_FormatString;
END_VAR
THIS^.assertorContainer.resetAssertor();

result := (valueToTest AND mask);
assertionIsWrong := (result = unexpected);
message := SEL(
	assertionIsWrong,
	'currentValue: 16#%.2X AND mask: 16#%.2X is 16#%.2X unexpectedValue: 16#%.2X assertion must be TRUE', 
	'currentValue: 16#%.2X AND mask: 16#%.2X is 16#%.2X unexpectedValue: 16#%.2X assertion must be FLASE'
);
messageStringBuilder(
	sFormat := message,
	arg1 := THIS^.AnyToArg(valueToTest),
	arg2 := THIS^.AnyToArg(mask),
	arg3 := THIS^.AnyToArg(result),
	arg4 := THIS^.AnyToArg(unexpected)
);


THIS^.assertorContainer.assertor.assert.bitNumber.short.andMaskIsNotEqualTo(
	currentValue	:= valueToTest,
	mask 			:= mask,
	unexpectedValue	:= unexpected,
	message			:= ''
);

THIS^.AssertEquals_BOOL(
	Expected 	:= assertionIsWrong,
	Actual 		:= THIS^.assertorContainer.wasAssertionWrong,
	Message 	:= messageStringBuilder.sOut
);
END_METHOD

(*

short summary
==================
This test method tests ``assert.bitNumber.short.bitXIsEqualTo``
method of CNM_AssertionInterfaces library, 
it provides the possibility to handover test data via parameter 


.. <legal notes>

legal notes
=================
| SPDX-FileCopyrightText: © 2022 ekvip automation GmbH <info@ekvip.de>
| SPDX-License-Identifier: Apache-2.0
| For details check: Apache-2.0_

.. _Apache-2.0: https://www.apache.org/licenses/LICENSE-2.0

.. </legal notes>

parameters
==========

*)

METHOD testBitXIsEqualTo
VAR_INPUT
	(* for the test it's the parameter ``currentValue`` *)
	valueToTest			:BYTE;
	(* the bit number to check in this test, it's the parameter ``number``*)
	bitNumberToCheck	:CNM_AssertionInterfaces.BitNumberByte;
	(* this is the expected value of the bit ``bitNumberToCheck``, it's the parameter ``expectedValue`` *)
	bitIsSet			:BOOL;
END_VAR
VAR
	(* just the expectation if the assertion to test must be worng or true *)
	assertionIsWrong		:BOOL;
	(* bit with the number of ``bitNumberToCheck`` filtered from ``valueToTest`` *)
	specificBitOnly			:BYTE;
	(* the bit number ``bitNumberToCheck`` is set to the value of ``bitIsSet`` only *)
	testBitOnly				:BYTE;
	(* contains the format string for the test message *)
	message					:Tc2_System.T_MaxString;
	(* TwinCAT printf with the test message *)
	messageStringBuilder	:Tc2_Utilities.FB_FormatString;
END_VAR
THIS^.assertorContainer.resetAssertor();

specificBitOnly := (valueToTest AND SHL(THIS^.LSB_ONLY,bitNumberToCheck));
testBitOnly		:= SHL(TO_BYTE(bitIsSet),bitNumberToCheck);
assertionIsWrong := (specificBitOnly <> testBitOnly);

message := 'Bit number %d in currentValue: 16#%.2X ';
message := SEL(
	(specificBitOnly > THIS^.NO_BIT_SET),
	Tc2_Standard.CONCAT(message, 'is unset '),
	Tc2_Standard.CONCAT(message, 'is set ')
);
message := SEL(
	(testBitOnly > THIS^.NO_BIT_SET),
	Tc2_Standard.CONCAT(message, 'expectedValue: is unset (FALSE) '),
	Tc2_Standard.CONCAT(message, 'expectedValue: is set (TRUE)  ')
);
message := SEL(
	assertionIsWrong,
	Tc2_Standard.CONCAT(message, 'assertion must be TRUE'),
	Tc2_Standard.CONCAT(message, 'assertion must be FALSE')
);
messageStringBuilder(
	sFormat := message,
	arg1 := THIS^.AnyToArg(bitNumberToCheck),
	arg2 := THIS^.AnyToArg(valueToTest)
);


THIS^.assertorContainer.assertor.assert.bitNumber.short.bitXIsEqualTo(
	currentValue 	:= valueToTest,
	number			:= bitNumberToCheck,
	expectedValue	:= bitIsSet,
	message			:= ''  
); 

THIS^.AssertEquals_BOOL(
	Expected 	:= assertionIsWrong,
	Actual 		:= THIS^.assertorContainer.wasAssertionWrong,
	Message 	:= messageStringBuilder.sOut
);
END_METHOD

(*

short summary
==================
This test method tests ``assert.bitNumber.short.bitXIsNotEqualTo``
method of CNM_AssertionInterfaces library, 
it provides the possibility to handover test data via parameter 


.. <legal notes>

legal notes
=================
| SPDX-FileCopyrightText: © 2022 ekvip automation GmbH <info@ekvip.de>
| SPDX-License-Identifier: Apache-2.0
| For details check: Apache-2.0_

.. _Apache-2.0: https://www.apache.org/licenses/LICENSE-2.0

.. </legal notes>

parameters
==========

*)

METHOD testBitXIsNotEqualTo
VAR_INPUT
	(* for the test it's the parameter ``currentValue`` *)
	valueToTest			:BYTE;
	(* the bit number to check in this test, it's the parameter ``number``*)
	bitNumberToCheck	:CNM_AssertionInterfaces.BitNumberByte;
	(* this is the unexpected value of the bit ``bitNumberToCheck``, it's the parameter ``unexpectedValue`` *)
	bitIsSet			:BOOL;
END_VAR
VAR
	(* just the expectation if the assertion to test must be worng or true *)
	assertionIsWrong		:BOOL;
	(* bit with the number of ``bitNumberToCheck`` filtered from ``valueToTest`` *)
	specificBitOnly			:BYTE;
	(* the bit number ``bitNumberToCheck`` is set to the value of ``bitIsSet`` only *)
	testBitOnly				:BYTE;
	(* contains the format string for the test message *)
	message					:Tc2_System.T_MaxString;
	(* TwinCAT printf with the test message *)
	messageStringBuilder	:Tc2_Utilities.FB_FormatString;
END_VAR
THIS^.assertorContainer.resetAssertor();

specificBitOnly := (valueToTest AND SHL(THIS^.LSB_ONLY,bitNumberToCheck));
testBitOnly		:= SHL(TO_BYTE(bitIsSet),bitNumberToCheck);
assertionIsWrong := (specificBitOnly = testBitOnly);

message := 'Bit number %d in currentValue: 16#%.2X ';
message := SEL(
	(specificBitOnly > THIS^.NO_BIT_SET),
	Tc2_Standard.CONCAT(message, 'is unset '),
	Tc2_Standard.CONCAT(message, 'is set ')
);
message := SEL(
	(testBitOnly > THIS^.NO_BIT_SET),
	Tc2_Standard.CONCAT(message, 'unexpectedValue: is unset (FALSE) '),
	Tc2_Standard.CONCAT(message, 'unexpectedValue: is set (TRUE)  ')
);
message := SEL(
	assertionIsWrong,
	Tc2_Standard.CONCAT(message, 'assertion must be TRUE'),
	Tc2_Standard.CONCAT(message, 'assertion must be FALSE')
);
messageStringBuilder(
	sFormat := message,
	arg1 := THIS^.AnyToArg(bitNumberToCheck),
	arg2 := THIS^.AnyToArg(valueToTest)
);

THIS^.assertorContainer.assertor.assert.bitNumber.short.bitXIsNotEqualTo(
	currentValue 	:= valueToTest,
	number			:= bitNumberToCheck,
	unexpectedValue	:= bitIsSet,
	message			:= ''  
); 

THIS^.AssertEquals_BOOL(
	Expected 	:= assertionIsWrong,
	Actual 		:= THIS^.assertorContainer.wasAssertionWrong,
	Message 	:= messageStringBuilder.sOut
);
END_METHOD

(*

short summary
==================
This test method tests ``assert.bitNumber.short.bitXIsSet``
of CNM_AssertionInterfaces library, 
it provides the possibility to handover test data via parameter 


.. <legal notes>

legal notes
=================
| SPDX-FileCopyrightText: © 2022 ekvip automation GmbH <info@ekvip.de>
| SPDX-License-Identifier: Apache-2.0
| For details check: Apache-2.0_

.. _Apache-2.0: https://www.apache.org/licenses/LICENSE-2.0

.. </legal notes>

parameters
==========

*)

METHOD testBitXIsSet
VAR_INPUT
	(* for the test it's the parameter ``currentValue`` *)
	valueToTest			:BYTE;
	(* the bit number to check in this test, it's the parameter ``number``*)
	bitNumberToCheck	:CNM_AssertionInterfaces.BitNumberByte;
END_VAR
VAR
	(* just the expectation if the assertion to test must be worng or true *)
	assertionIsWrong		:BOOL;
	(* contains the format string for the test message *)
	message					:Tc2_System.T_MaxString;
	(* TwinCAT printf with the test message *)
	messageStringBuilder	:Tc2_Utilities.FB_FormatString;
END_VAR
THIS^.assertorContainer.resetAssertor();

assertionIsWrong := ((valueToTest AND SHL(THIS^.LSB_ONLY,bitNumberToCheck)) = THIS^.NO_BIT_SET);

message := SEL(
	assertionIsWrong,
	'Bit number %d in currentValue: 16#%.2X is set assertion must be TRUE',
	'Bit number %d in currentValue: 16#%.2X is unset assertion must be FALSE'
);

messageStringBuilder(
	sFormat := message,
	arg1 := THIS^.AnyToArg(bitNumberToCheck),
	arg2 := THIS^.AnyToArg(valueToTest)
);

THIS^.assertorContainer.assertor.assert.bitNumber.short.bitXIsSet(
	currentValue := valueToTest,
	number := bitNumberToCheck,
	message := ''
);

THIS^.AssertEquals_BOOL(
	Expected 	:= assertionIsWrong,
	Actual 		:= THIS^.assertorContainer.wasAssertionWrong,
	Message 	:= messageStringBuilder.sOut
);
END_METHOD

(*

short summary
==================
This test method tests ``assert.bitNumber.short.bitXIsUnset``
of CNM_AssertionInterfaces library, 
it provides the possibility to handover test data via parameter 


.. <legal notes>

legal notes
=================
| SPDX-FileCopyrightText: © 2022 ekvip automation GmbH <info@ekvip.de>
| SPDX-License-Identifier: Apache-2.0
| For details check: Apache-2.0_

.. _Apache-2.0: https://www.apache.org/licenses/LICENSE-2.0

.. </legal notes>

parameters
==========

*)

METHOD testBitXIsUnset
VAR_INPUT
	(* for the test it's the parameter ``currentValue`` *)
	valueToTest			:BYTE;
	(* the bit number to check in this test, it's the parameter ``number``*)
	bitNumberToCheck	:CNM_AssertionInterfaces.BitNumberByte;
END_VAR
VAR
	(* just the expectation if the assertion to test must be worng or true *)
	assertionIsWrong		:BOOL;
	(* contains the format string for the test message *)
	message					:Tc2_System.T_MaxString;
	(* TwinCAT printf with the test message *)
	messageStringBuilder	:Tc2_Utilities.FB_FormatString;
END_VAR
THIS^.assertorContainer.resetAssertor();

assertionIsWrong := ((valueToTest AND SHL(THIS^.LSB_ONLY,bitNumberToCheck)) > THIS^.NO_BIT_SET);

message := SEL(
	assertionIsWrong,
	'Bit number %d in currentValue: 16#%.2X is unset assertion must be TRUE',
	'Bit number %d in currentValue: 16#%.2X is set assertion must be FALSE'
);

messageStringBuilder(
	sFormat := message,
	arg1 := THIS^.AnyToArg(bitNumberToCheck),
	arg2 := THIS^.AnyToArg(valueToTest)
);

THIS^.assertorContainer.assertor.assert.bitNumber.short.bitXIsUnset(
	currentValue := valueToTest,
	number := bitNumberToCheck,
	message := ''
);

THIS^.AssertEquals_BOOL(
	Expected 	:= assertionIsWrong,
	Actual 		:= THIS^.assertorContainer.wasAssertionWrong,
	Message 	:= messageStringBuilder.sOut
);
END_METHOD

(*

short summary
==================
This test method tests ``assert.bitNumber.short.lsbIsEqualTo``
method of CNM_AssertionInterfaces library, 
it provides the possibility to handover test data via parameter 


.. <legal notes>

legal notes
=================
| SPDX-FileCopyrightText: © 2022 ekvip automation GmbH <info@ekvip.de>
| SPDX-License-Identifier: Apache-2.0
| For details check: Apache-2.0_

.. _Apache-2.0: https://www.apache.org/licenses/LICENSE-2.0

.. </legal notes>

parameters
==========

*)

METHOD testLsbIsEqualTo
VAR_INPUT
	(* for the test it's the parameter ``currentValue`` *)
	valueToTest		:BYTE;
	(* for the test it's the parameter ``expectedValue`` *)
	expectedValue	:BOOL;
END_VAR
VAR
	(* just the expectation if the assertion to test must be worng or true *)
	assertionIsWrong		:BOOL;
	(* contains the format string for the test message *)
	message					:Tc2_System.T_MaxString;
	(* TwinCAT printf with the test message *)
	messageStringBuilder	:Tc2_Utilities.FB_FormatString;
END_VAR
THIS^.assertorContainer.resetAssertor();

assertionIsWrong := (valueToTest.FIRST_BIT <> expectedValue);
message := SEL(
	expectedValue,
	'currentValue: %d expectedValue is an unset (FALSE) assertion must be ',
	'currentValue: %d expectedValue is a set (TRUE) assertion must be '
);
message := SEL(
	assertionIsWrong,
	Tc2_Standard.CONCAT(message, 'TRUE'),
	Tc2_Standard.CONCAT(message, 'FALSE')
);

messageStringBuilder(
	sFormat := message,
	arg1 := THIS^.AnyToArg(valueToTest)
);

THIS^.assertorContainer.assertor.assert.bitNumber.short.lsbIsEqualTo(
	currentValue 	:= valueToTest,
	expectedValue	:= expectedValue,
	message			:= ''  
); 

THIS^.AssertEquals_BOOL(
	Expected 	:= assertionIsWrong,
	Actual 		:= THIS^.assertorContainer.wasAssertionWrong,
	Message 	:= messageStringBuilder.sOut
);
END_METHOD

(*

short summary
==================
This test method tests ``assert.bitNumber.short.lsbIsNotEqualTo``
method of CNM_AssertionInterfaces library, 
it provides the possibility to handover test data via parameter 


.. <legal notes>

legal notes
=================
| SPDX-FileCopyrightText: © 2022 ekvip automation GmbH <info@ekvip.de>
| SPDX-License-Identifier: Apache-2.0
| For details check: Apache-2.0_

.. _Apache-2.0: https://www.apache.org/licenses/LICENSE-2.0

.. </legal notes>

parameters
==========

*)

METHOD testLsbIsNotEqualTo
VAR_INPUT
	(* for the test it's the parameter ``currentValue`` *)
	valueToTest	:BYTE;
	(* for the test it's the parameter ``unexpectedValue`` *)
	unexpectedValue :BOOL;
END_VAR
VAR
	(* just the expectation if the assertion to test must be worng or true *)
	assertionIsWrong		:BOOL;
	(* contains the format string for the test message *)
	message					:Tc2_System.T_MaxString;
	(* TwinCAT printf with the test message *)
	messageStringBuilder	:Tc2_Utilities.FB_FormatString;
END_VAR
THIS^.assertorContainer.resetAssertor();

assertionIsWrong := (valueToTest.FIRST_BIT = unexpectedValue);
message := SEL(
	unexpectedValue,
	'currentValue: %d unexpectedValue is an unset (FALSE), assertion must be ',
	'currentValue: %d unexpectedValue is a set (TRUE) assertion must be '
);
message := SEL(
	assertionIsWrong,
	Tc2_Standard.CONCAT(message, 'TRUE'),
	Tc2_Standard.CONCAT(message, 'FALSE')
);

messageStringBuilder(
	sFormat := message,
	arg1 := THIS^.AnyToArg(valueToTest)
);

THIS^.assertorContainer.assertor.assert.bitNumber.short.lsbIsNotEqualTo(
	currentValue 	:= valueToTest,
	unexpectedValue	:= unexpectedValue,
	message			:= ''  
); 

THIS^.AssertEquals_BOOL(
	Expected 	:= assertionIsWrong,
	Actual 		:= THIS^.assertorContainer.wasAssertionWrong,
	Message 	:= messageStringBuilder.sOut
);
END_METHOD

(*

short summary
==================
This test method tests ``assert.bitNumber.short.lsbIsSet``
of CNM_AssertionInterfaces library, 
it provides the possibility to handover test data via parameter 


.. <legal notes>

legal notes
=================
| SPDX-FileCopyrightText: © 2022 ekvip automation GmbH <info@ekvip.de>
| SPDX-License-Identifier: Apache-2.0
| For details check: Apache-2.0_

.. _Apache-2.0: https://www.apache.org/licenses/LICENSE-2.0

.. </legal notes>

parameters
==========

*)

METHOD testLsbIsSet
VAR_INPUT
	(* for the test it's the parameter ``currentValue`` *)
	valueToTest	:BYTE;
END_VAR
VAR
	(* just the expectation if the assertion to test must be worng or true *)
	assertionIsWrong		:BOOL;
	(* contains the format string for the test message *)
	message					:Tc2_System.T_MaxString;
	(* TwinCAT printf with the test message *)
	messageStringBuilder	:Tc2_Utilities.FB_FormatString;
END_VAR
THIS^.assertorContainer.resetAssertor();

assertionIsWrong := (NOT valueToTest.FIRST_BIT);

message := SEL(
	assertionIsWrong,
	'currentValue is %d assertion must be TRUE',
	'currentValue is %d assertion must be FALSE'
);

messageStringBuilder(
	sFormat := message,
	arg1 := THIS^.AnyToArg(valueToTest)
);

THIS^.assertorContainer.assertor.assert.bitNumber.short.lsbIsSet(
	currentValue 	:= valueToTest,
	message			:= ''  
); 

THIS^.AssertEquals_BOOL(
	Expected 	:= assertionIsWrong,
	Actual 		:= THIS^.assertorContainer.wasAssertionWrong,
	Message 	:= messageStringBuilder.sOut
);
END_METHOD

(*

short summary
==================
This test method tests ``assert.bitNumber.short.lsbIsUnset``
and ``assert.bitNumber.short.lsbIsUnset``
of CNM_AssertionInterfaces library, 
it provides the possibility to handover test data via parameter 


.. <legal notes>

legal notes
=================
| SPDX-FileCopyrightText: © 2022 ekvip automation GmbH <info@ekvip.de>
| SPDX-License-Identifier: Apache-2.0
| For details check: Apache-2.0_

.. _Apache-2.0: https://www.apache.org/licenses/LICENSE-2.0

.. </legal notes>

parameters
==========

*)

METHOD testLsbIsUnset
VAR_INPUT
	(* for the test it's the parameter ``currentValue`` *)
	valueToTest	:BYTE;
END_VAR
VAR
	(* just the expectation if the assertion to test must be worng or true *)
	assertionIsWrong		:BOOL;
	(* contains the format string for the test message *)
	message					:Tc2_System.T_MaxString;
	(* TwinCAT printf with the test message *)
	messageStringBuilder	:Tc2_Utilities.FB_FormatString;
END_VAR
THIS^.assertorContainer.resetAssertor();

assertionIsWrong := (valueToTest.FIRST_BIT);

message := SEL(
	assertionIsWrong,
	'currentValue is %d assertion must be TRUE',
	'currentValue is %d assertion must be FALSE'
);

messageStringBuilder(
	sFormat := message,
	arg1 := THIS^.AnyToArg(valueToTest)
);

THIS^.assertorContainer.assertor.assert.bitNumber.short.lsbIsUnset(
	currentValue 	:= valueToTest,
	message			:= ''  
); 

THIS^.AssertEquals_BOOL(
	Expected 	:= assertionIsWrong,
	Actual 		:= THIS^.assertorContainer.wasAssertionWrong,
	Message 	:= messageStringBuilder.sOut
);
END_METHOD

(*

short summary
==================
This test method tests ``assert.bitNumber.short.msbIsEqualTo``
method of CNM_AssertionInterfaces library, 
it provides the possibility to handover test data via parameter 


.. <legal notes>

legal notes
=================
| SPDX-FileCopyrightText: © 2022 ekvip automation GmbH <info@ekvip.de>
| SPDX-License-Identifier: Apache-2.0
| For details check: Apache-2.0_

.. _Apache-2.0: https://www.apache.org/licenses/LICENSE-2.0

.. </legal notes>

parameters
==========

*)

METHOD testMsbIsEqualTo
VAR_INPUT
	(* for the test it's the parameter ``currentValue`` *)
	valueToTest		:BYTE;
	(* for the test it's the parameter ``expectedValue`` *)
	expectedValue	:BOOL;
END_VAR
VAR
	(* just the expectation if the assertion to test must be worng or true *)
	assertionIsWrong		:BOOL;
	(* contains the format string for the test message *)
	message					:Tc2_System.T_MaxString;
	(* TwinCAT printf with the test message *)
	messageStringBuilder	:Tc2_Utilities.FB_FormatString;
END_VAR
THIS^.assertorContainer.resetAssertor();

assertionIsWrong := (valueToTest.LAST_BIT <> expectedValue);

message := SEL(
	expectedValue,
	'currentValue: 16#%.2X expectedValue is an unset (FALSE) assertion must be ',
	'currentValue: 16#%.2X expectedValue is a set (TRUE) assertion must be '
);
message := SEL(
	assertionIsWrong,
	Tc2_Standard.CONCAT(message, 'TRUE'),
	Tc2_Standard.CONCAT(message, 'FALSE')
);

messageStringBuilder(
	sFormat := message,
	arg1 := THIS^.AnyToArg(valueToTest)
);

THIS^.assertorContainer.assertor.assert.bitNumber.short.msbIsEqualTo(
	currentValue 	:= valueToTest,
	expectedValue	:= expectedValue,
	message			:= ''  
); 

THIS^.AssertEquals_BOOL(
	Expected 	:= assertionIsWrong,
	Actual 		:= THIS^.assertorContainer.wasAssertionWrong,
	Message 	:= messageStringBuilder.sOut
);
END_METHOD

(*

short summary
==================
This test method tests ``assert.bitNumber.short.msbIsNotEqualTo``
method of CNM_AssertionInterfaces library, 
it provides the possibility to handover test data via parameter 


.. <legal notes>

legal notes
=================
| SPDX-FileCopyrightText: © 2022 ekvip automation GmbH <info@ekvip.de>
| SPDX-License-Identifier: Apache-2.0
| For details check: Apache-2.0_

.. _Apache-2.0: https://www.apache.org/licenses/LICENSE-2.0

.. </legal notes>

parameters
==========

*)

METHOD testMsbIsNotEqualTo
VAR_INPUT
	(* for the test it's the parameter ``currentValue`` *)
	valueToTest	:BYTE;
	(* for the test it's the parameter ``unexpectedValue`` *)
	unexpectedValue :BOOL;
END_VAR
VAR
	(* just the expectation if the assertion to test must be worng or true *)
	assertionIsWrong		:BOOL;
	(* contains the format string for the test message *)
	message					:Tc2_System.T_MaxString;
	(* TwinCAT printf with the test message *)
	messageStringBuilder	:Tc2_Utilities.FB_FormatString;
END_VAR
THIS^.assertorContainer.resetAssertor();

assertionIsWrong := (valueToTest.LAST_BIT = unexpectedValue);

